LIN {X 0,Y 574.132,Z 514.669,A -85,B 0,C 180,E1 -2084.662,E2 -2084.662} C_VEL
LIN {X 0,Y 574.281,Z 500.292,A -85,B 0,C 180,E1 -2084.996,E2 -2084.996} C_VEL
LIN {X 0,Y 573.065,Z 493.165,A -85,B 0,C 180,E1 -2085.151,E2 -2085.151} C_VEL
LIN {X 0,Y 573.135,Z 485.279,A -85,B 0,C 180,E1 -2087.851,E2 -2087.851} C_VEL
LIN {X 0,Y 573.19,Z 477.793,A -85,B 0,C 180,E1 -2090.452,E2 -2090.452} C_VEL
LIN {X 0,Y 573.212,Z 470.196,A -85,B 0,C 180,E1 -2093.139,E2 -2093.139} C_VEL
LIN {X 0,Y 573.285,Z 462.82,A -85,B 0,C 180,E1 -2095.797,E2 -2095.797} C_VEL
LIN {X 0,Y 573.314,Z 455.113,A -85,B 0,C 180,E1 -2098.559,E2 -2098.559} C_VEL
LIN {X 0,Y 573.308,Z 448.157,A -85,B 0,C 180,E1 -2100.987,E2 -2100.987} C_VEL
LIN {X 0,Y 573.317,Z 439.853,A -85,B 0,C 180,E1 -2103.899,E2 -2103.899} C_VEL
LIN {X 0,Y 573.354,Z 431.271,A -85,B 0,C 180,E1 -2106.913,E2 -2106.913} C_VEL
LIN {X 0,Y 573.295,Z 427.699,A -85,B 0,C 180,E1 -2108.186,E2 -2108.186} C_VEL
LIN {X 0,Y 573.264,Z 427.702,A -85,B 0,C 180,E1 -2110.527,E2 -2110.527} C_VEL
LIN {X 0,Y 573.246,Z 427.701,A -85,B 0,C 180,E1 -2113.669,E2 -2113.669} C_VEL
LIN {X 0,Y 573.247,Z 427.703,A -85,B 0,C 180,E1 -2116.641,E2 -2116.641} C_VEL
LIN {X 0,Y 573.267,Z 427.705,A -85,B 0,C 180,E1 -2119.477,E2 -2119.477} C_VEL
LIN {X 0,Y 573.23,Z 427.703,A -85,B 0,C 180,E1 -2122.192,E2 -2122.192} C_VEL
LIN {X 0,Y 573.26,Z 427.706,A -85,B 0,C 180,E1 -2124.816,E2 -2124.816} C_VEL
LIN {X 0,Y 573.25,Z 427.701,A -85,B 0,C 180,E1 -2127.355,E2 -2127.355} C_VEL
LIN {X 0,Y 573.248,Z 427.705,A -85,B 0,C 180,E1 -2129.824,E2 -2129.824} C_VEL
LIN {X 0,Y 573.28,Z 427.697,A -85,B 0,C 180,E1 -2132.234,E2 -2132.234} C_VEL
LIN {X 0,Y 573.26,Z 427.706,A -85,B 0,C 180,E1 -2135.12,E2 -2135.12} C_VEL
LIN {X 0,Y 573.25,Z 427.699,A -85,B 0,C 180,E1 -2137.663,E2 -2137.663} C_VEL
LIN {X 0,Y 573.27,Z 427.701,A -85,B 0,C 180,E1 -2140.727,E2 -2140.727} C_VEL
LIN {X 0,Y 573.252,Z 427.704,A -85,B 0,C 180,E1 -2143.622,E2 -2143.622} C_VEL
LIN {X 0,Y 573.23,Z 427.703,A -85,B 0,C 180,E1 -2146.529,E2 -2146.529} C_VEL
LIN {X 0,Y 573.273,Z 427.7,A -85,B 0,C 180,E1 -2148.734,E2 -2148.734} C_VEL
LIN {X 0,Y 573.3,Z 427.693,A -85,B 0,C 180,E1 -2151.541,E2 -2151.541} C_VEL
LIN {X 0,Y 573.295,Z 427.7,A -85,B 0,C 180,E1 -2154.372,E2 -2154.372} C_VEL
LIN {X 0,Y 573.3,Z 427.698,A -85,B 0,C 180,E1 -2157.892,E2 -2157.892} C_VEL
LIN {X 0,Y 573.328,Z 427.692,A -85,B 0,C 180,E1 -2160.702,E2 -2160.702} C_VEL
LIN {X 0,Y 573.236,Z 427.699,A -85,B 0,C 180,E1 -2163.514,E2 -2163.514} C_VEL
LIN {X 0,Y 573.287,Z 427.695,A -85,B 0,C 180,E1 -2165.628,E2 -2165.628} C_VEL
LIN {X 0,Y 573.3,Z 427.696,A -85,B 0,C 180,E1 -2168.459,E2 -2168.459} C_VEL
LIN {X 0,Y 573.288,Z 427.696,A -85,B 0,C 180,E1 -2171.312,E2 -2171.312} C_VEL
LIN {X 0,Y 573.271,Z 427.698,A -85,B 0,C 180,E1 -2174.425,E2 -2174.425} C_VEL
LIN {X 0,Y 573.251,Z 427.7,A -85,B 0,C 180,E1 -2177.112,E2 -2177.112} C_VEL
LIN {X 0,Y 573.249,Z 427.705,A -85,B 0,C 180,E1 -2180.077,E2 -2180.077} C_VEL
LIN {X 0,Y 573.234,Z 427.705,A -85,B 0,C 180,E1 -2182.338,E2 -2182.338} C_VEL
LIN {X 0,Y 573.248,Z 427.708,A -85,B 0,C 180,E1 -2185.41,E2 -2185.41} C_VEL
LIN {X 0,Y 573.256,Z 427.699,A -85,B 0,C 180,E1 -2188.033,E2 -2188.033} C_VEL
LIN {X 0,Y 573.237,Z 427.706,A -85,B 0,C 180,E1 -2190.886,E2 -2190.886} C_VEL
LIN {X 0,Y 573.279,Z 427.698,A -85,B 0,C 180,E1 -2193.529,E2 -2193.529} C_VEL
LIN {X 0,Y 573.253,Z 427.704,A -85,B 0,C 180,E1 -2196.049,E2 -2196.049} C_VEL
LIN {X 0,Y 573.242,Z 427.702,A -85,B 0,C 180,E1 -2198.702,E2 -2198.702} C_VEL
LIN {X 0,Y 573.259,Z 427.7,A -85,B 0,C 180,E1 -2201.598,E2 -2201.598} C_VEL
LIN {X 0,Y 573.232,Z 427.708,A -85,B 0,C 180,E1 -2204.334,E2 -2204.334} C_VEL
LIN {X 0,Y 573.234,Z 427.703,A -85,B 0,C 180,E1 -2207.359,E2 -2207.359} C_VEL
LIN {X 0,Y 573.245,Z 427.702,A -85,B 0,C 180,E1 -2210.394,E2 -2210.394} C_VEL
LIN {X 0,Y 573.251,Z 427.707,A -85,B 0,C 180,E1 -2213.079,E2 -2213.079} C_VEL
LIN {X 0,Y 573.271,Z 427.701,A -85,B 0,C 180,E1 -2215.673,E2 -2215.673} C_VEL
LIN {X 0,Y 573.301,Z 427.855,A -85,B 0,C 180,E1 -2216.679,E2 -2216.679} C_VEL
LIN {X 0,Y 573.955,Z 432.32,A -85,B 0,C 180,E1 -2217.952,E2 -2217.952} C_VEL
LIN {X 0,Y 573.773,Z 442.67,A -85,B 0,C 180,E1 -2220.664,E2 -2220.664} C_VEL
LIN {X 0,Y 573.669,Z 453.5,A -85,B 0,C 180,E1 -2223.421,E2 -2223.421} C_VEL
LIN {X 0,Y 573.507,Z 464.501,A -85,B 0,C 180,E1 -2226.148,E2 -2226.148} C_VEL
LIN {X 0,Y 573.373,Z 476.989,A -85,B 0,C 180,E1 -2229.179,E2 -2229.179} C_VEL
LIN {X 0,Y 573.305,Z 489.478,A -85,B 0,C 180,E1 -2232.155,E2 -2232.155} C_VEL
LIN {X 0,Y 573.22,Z 501.089,A -85,B 0,C 180,E1 -2234.876,E2 -2234.876} C_VEL
LIN {X 0,Y 574.273,Z 507.817,A -85,B 0,C 180,E1 -2235.005,E2 -2235.005} C_VEL
LIN {X 0,Y 574.185,Z 522.276,A -85,B 0,C 180,E1 -2235.316,E2 -2235.316} C_VEL
LIN {X 0,Y 574.055,Z 536.338,A -85,B 0,C 180,E1 -2235.772,E2 -2235.772} C_VEL
LIN {X 0,Y 573.93,Z 549.901,A -85,B 0,C 180,E1 -2236.367,E2 -2236.367} C_VEL
LIN {X 0,Y 573.716,Z 562.7,A -85,B 0,C 180,E1 -2237.083,E2 -2237.083} C_VEL
LIN {X 0,Y 573.571,Z 575.491,A -85,B 0,C 180,E1 -2237.978,E2 -2237.978} C_VEL
LIN {X 0,Y 573.448,Z 586.864,A -85,B 0,C 180,E1 -2238.956,E2 -2238.956} C_VEL
LIN {X 0,Y 573.268,Z 596.342,A -85,B 0,C 180,E1 -2239.94,E2 -2239.94} C_VEL
LIN {X 0,Y 573.19,Z 604.92,A -85,B 0,C 180,E1 -2241.007,E2 -2241.007} C_VEL
LIN {X 0,Y 573.111,Z 613.121,A -85,B 0,C 180,E1 -2242.249,E2 -2242.249} C_VEL
LIN {X 0,Y 573.035,Z 619.452,A -85,B 0,C 180,E1 -2243.427,E2 -2243.427} C_VEL
LIN {X 0,Y 573.001,Z 624.965,A -85,B 0,C 180,E1 -2244.723,E2 -2244.723} C_VEL
LIN {X 0,Y 573.028,Z 628.445,A -85,B 0,C 180,E1 -2245.781,E2 -2245.781} C_VEL
LIN {X 0,Y 572.956,Z 631.833,A -85,B 0,C 180,E1 -2247.189,E2 -2247.189} C_VEL
LIN {X 0,Y 572.941,Z 633.833,A -85,B 0,C 180,E1 -2248.595,E2 -2248.595} C_VEL
LIN {X 0,Y 572.937,Z 634.5,A -85,B 0,C 180,E1 -2250.001,E2 -2250.001} C_VEL
LIN {X 0,Y 572.941,Z 633.832,A -85,B 0,C 180,E1 -2251.407,E2 -2251.407} C_VEL
LIN {X 0,Y 572.956,Z 631.831,A -85,B 0,C 180,E1 -2252.813,E2 -2252.813} C_VEL
LIN {X 0,Y 573.028,Z 628.441,A -85,B 0,C 180,E1 -2254.221,E2 -2254.221} C_VEL
LIN {X 0,Y 573.055,Z 623.564,A -85,B 0,C 180,E1 -2255.631,E2 -2255.631} C_VEL
LIN {X 0,Y 573.059,Z 618.849,A -85,B 0,C 180,E1 -2256.693,E2 -2256.693} C_VEL
LIN {X 0,Y 573.126,Z 612.032,A -85,B 0,C 180,E1 -2257.93,E2 -2257.93} C_VEL
LIN {X 0,Y 573.226,Z 603.553,A -85,B 0,C 180,E1 -2259.172,E2 -2259.172} C_VEL
LIN {X 0,Y 573.305,Z 594.7,A -85,B 0,C 180,E1 -2260.24,E2 -2260.24} C_VEL
LIN {X 0,Y 573.464,Z 583.983,A -85,B 0,C 180,E1 -2261.309,E2 -2261.309} C_VEL
LIN {X 0,Y 573.622,Z 573.133,A -85,B 0,C 180,E1 -2262.202,E2 -2262.202} C_VEL
LIN {X 0,Y 573.736,Z 561.247,A -85,B 0,C 180,E1 -2263.009,E2 -2263.009} C_VEL
LIN {X 0,Y 573.95,Z 548.078,A -85,B 0,C 180,E1 -2263.725,E2 -2263.725} C_VEL
LIN {X 0,Y 574.08,Z 534.798,A -85,B 0,C 180,E1 -2264.285,E2 -2264.285} C_VEL
LIN {X 0,Y 574.206,Z 520.732,A -85,B 0,C 180,E1 -2264.722,E2 -2264.722} C_VEL
LIN {X 0,Y 574.197,Z 506.39,A -85,B 0,C 180,E1 -2265.019,E2 -2265.019} C_VEL
LIN {X 0,Y 573.209,Z 501.081,A -85,B 0,C 180,E1 -2265.126,E2 -2265.126} C_VEL
LIN {X 0,Y 573.307,Z 489.47,A -85,B 0,C 180,E1 -2267.847,E2 -2267.847} C_VEL
LIN {X 0,Y 573.373,Z 476.982,A -85,B 0,C 180,E1 -2270.822,E2 -2270.822} C_VEL
LIN {X 0,Y 573.516,Z 465.991,A -85,B 0,C 180,E1 -2273.486,E2 -2273.486} C_VEL
LIN {X 0,Y 573.613,Z 455.126,A -85,B 0,C 180,E1 -2276.173,E2 -2276.173} C_VEL
LIN {X 0,Y 573.767,Z 445.866,A -85,B 0,C 180,E1 -2278.536,E2 -2278.536} C_VEL
LIN {X 0,Y 573.946,Z 436.55,A -85,B 0,C 180,E1 -2281.001,E2 -2281.001} C_VEL
LIN {X 0,Y 574.002,Z 431.778,A -85,B 0,C 180,E1 -2282.347,E2 -2282.347} C_VEL
LIN {X 0,Y 573.275,Z 427.703,A -85,B 0,C 180,E1 -2283.693,E2 -2283.693} C_VEL
LIN {X 0,Y 573.244,Z 427.708,A -85,B 0,C 180,E1 -2286.05,E2 -2286.05} C_VEL
LIN {X 0,Y 573.253,Z 427.705,A -85,B 0,C 180,E1 -2288.701,E2 -2288.701} C_VEL
LIN {X 0,Y 573.233,Z 427.707,A -85,B 0,C 180,E1 -2291.458,E2 -2291.458} C_VEL
LIN {X 0,Y 573.229,Z 427.707,A -85,B 0,C 180,E1 -2294.335,E2 -2294.335} C_VEL
LIN {X 0,Y 573.252,Z 427.705,A -85,B 0,C 180,E1 -2296.642,E2 -2296.642} C_VEL
LIN {X 0,Y 573.249,Z 427.707,A -85,B 0,C 180,E1 -2299.475,E2 -2299.475} C_VEL
LIN {X 0,Y 573.239,Z 427.71,A -85,B 0,C 180,E1 -2302.193,E2 -2302.193} C_VEL
LIN {X 0,Y 573.313,Z 427.8,A -85,B 0,C 180,E1 -2304.551,E2 -2304.551} C_VEL
LIN {X 0,Y 573.264,Z 433.787,A -85,B 0,C 180,E1 -2307.356,E2 -2307.356} C_VEL
LIN {X 0,Y 573.239,Z 440.605,A -85,B 0,C 180,E1 -2310.514,E2 -2310.514} C_VEL
LIN {X 0,Y 573.167,Z 446.058,A -85,B 0,C 180,E1 -2313.02,E2 -2313.02} C_VEL
LIN {X 0,Y 573.161,Z 451.002,A -85,B 0,C 180,E1 -2315.361,E2 -2315.361} C_VEL
LIN {X 0,Y 573.094,Z 457.867,A -85,B 0,C 180,E1 -2318.414,E2 -2318.414} C_VEL
LIN {X 0,Y 573.064,Z 464.731,A -85,B 0,C 180,E1 -2321.406,E2 -2321.406} C_VEL
LIN {X 0,Y 573.047,Z 469.879,A -85,B 0,C 180,E1 -2323.616,E2 -2323.616} C_VEL
LIN {X 0,Y 573.049,Z 475.028,A -85,B 0,C 180,E1 -2325.801,E2 -2325.801} C_VEL
LIN {X 0,Y 573.015,Z 479.212,A -85,B 0,C 180,E1 -2327.561,E2 -2327.561} C_VEL
LIN {X 0,Y 573.855,Z 486.016,A -85,B 0,C 180,E1 -2327.714,E2 -2327.714} C_VEL
LIN {X 0,Y 573.738,Z 498.671,A -85,B 0,C 180,E1 -2328.071,E2 -2328.071} C_VEL
LIN {X 0,Y 573.604,Z 511.366,A -85,B 0,C 180,E1 -2328.578,E2 -2328.578} C_VEL
LIN {X 0,Y 573.544,Z 522.177,A -85,B 0,C 180,E1 -2329.147,E2 -2329.147} C_VEL
LIN {X 0,Y 573.441,Z 532.835,A -85,B 0,C 180,E1 -2329.853,E2 -2329.853} C_VEL
LIN {X 0,Y 573.321,Z 542.609,A -85,B 0,C 180,E1 -2330.652,E2 -2330.652} C_VEL
LIN {X 0,Y 573.235,Z 551.501,A -85,B 0,C 180,E1 -2331.54,E2 -2331.54} C_VEL
LIN {X 0,Y 573.126,Z 560.184,A -85,B 0,C 180,E1 -2332.602,E2 -2332.602} C_VEL
LIN {X 0,Y 573.049,Z 567.111,A -85,B 0,C 180,E1 -2333.663,E2 -2333.663} C_VEL
LIN {X 0,Y 573.009,Z 572.659,A -85,B 0,C 180,E1 -2334.722,E2 -2334.722} C_VEL
LIN {X 0,Y 573.031,Z 577.019,A -85,B 0,C 180,E1 -2335.78,E2 -2335.78} C_VEL
LIN {X 0,Y 573.023,Z 579.323,A -85,B 0,C 180,E1 -2336.484,E2 -2336.484} C_VEL
LIN {X 0,Y 572.959,Z 581.2,A -85,B 0,C 180,E1 -2337.188,E2 -2337.188} C_VEL
LIN {X 0,Y 572.938,Z 582.628,A -85,B 0,C 180,E1 -2337.891,E2 -2337.891} C_VEL
LIN {X 0,Y 572.941,Z 584.255,A -85,B 0,C 180,E1 -2339.297,E2 -2339.297} C_VEL
LIN {X 0,Y 572.938,Z 584.496,A -85,B 0,C 180,E1 -2340,E2 -2340} C_VEL
LIN {X 0,Y 572.941,Z 584.314,A -85,B 0,C 180,E1 -2340.703,E2 -2340.703} C_VEL
LIN {X 0,Y 572.937,Z 582.771,A -85,B 0,C 180,E1 -2342.109,E2 -2342.109} C_VEL
LIN {X 0,Y 572.96,Z 581.409,A -85,B 0,C 180,E1 -2342.812,E2 -2342.812} C_VEL
LIN {X 0,Y 573.015,Z 578.532,A -85,B 0,C 180,E1 -2343.868,E2 -2343.868} C_VEL
LIN {X 0,Y 572.963,Z 574.631,A -85,B 0,C 180,E1 -2344.926,E2 -2344.926} C_VEL
LIN {X 0,Y 573.073,Z 569.599,A -85,B 0,C 180,E1 -2345.984,E2 -2345.984} C_VEL
LIN {X 0,Y 573.084,Z 563.275,A -85,B 0,C 180,E1 -2347.044,E2 -2347.044} C_VEL
LIN {X 0,Y 573.175,Z 555.354,A -85,B 0,C 180,E1 -2348.106,E2 -2348.106} C_VEL
LIN {X 0,Y 573.287,Z 545.505,A -85,B 0,C 180,E1 -2349.17,E2 -2349.17} C_VEL
LIN {X 0,Y 573.412,Z 535.182,A -85,B 0,C 180,E1 -2350.059,E2 -2350.059} C_VEL
LIN {X 0,Y 573.509,Z 523.592,A -85,B 0,C 180,E1 -2350.857,E2 -2350.857} C_VEL
LIN {X 0,Y 573.642,Z 512.017,A -85,B 0,C 180,E1 -2351.482,E2 -2351.482} C_VEL
LIN {X 0,Y 573.729,Z 500.106,A -85,B 0,C 180,E1 -2351.97,E2 -2351.97} C_VEL
LIN {X 0,Y 573.859,Z 486.938,A -85,B 0,C 180,E1 -2352.353,E2 -2352.353} C_VEL
LIN {X 0,Y 573.47,Z 482.233,A -85,B 0,C 180,E1 -2352.461,E2 -2352.461} C_VEL
LIN {X 0,Y 573.01,Z 479.211,A -85,B 0,C 180,E1 -2352.529,E2 -2352.529} C_VEL
LIN {X 0,Y 573.05,Z 473.524,A -85,B 0,C 180,E1 -2354.925,E2 -2354.925} C_VEL
LIN {X 0,Y 573.062,Z 466.656,A -85,B 0,C 180,E1 -2357.854,E2 -2357.854} C_VEL
LIN {X 0,Y 573.069,Z 463.772,A -85,B 0,C 180,E1 -2359.099,E2 -2359.099} C_VEL
LIN {X 0,Y 572.427,Z 462.503,A -85,B 0,C 180,E1 -2359.672,E2 -2359.672} C_VEL
LIN {X 0,Y 569.575,Z 460.607,A -85,B 0,C 180,E1 -2360.606,E2 -2360.606} C_VEL
LIN {X 0,Y 567.148,Z 459.117,A -85,B 0,C 180,E1 -2361.358,E2 -2361.358} C_VEL
LIN {X 0,Y 566.103,Z 457.91,A -85,B 0,C 180,E1 -2361.938,E2 -2361.938} C_VEL
LIN {X 0,Y 566.017,Z 457.48,A -85,B 0,C 180,E1 -2362.133,E2 -2362.133} C_VEL
LIN {X 0,Y 566.079,Z 451.198,A -85,B 0,C 180,E1 -2364.999,E2 -2364.999} C_VEL
LIN {X 0,Y 566.104,Z 446.133,A -85,B 0,C 180,E1 -2367.345,E2 -2367.345} C_VEL
LIN {X 0,Y 566.17,Z 440.975,A -85,B 0,C 180,E1 -2369.771,E2 -2369.771} C_VEL
LIN {X 0,Y 566.218,Z 435.4,A -85,B 0,C 180,E1 -2372.431,E2 -2372.431} C_VEL
LIN {X 0,Y 566.268,Z 430.126,A -85,B 0,C 180,E1 -2375.001,E2 -2375.001} C_VEL
LIN {X 0,Y 566.25,Z 428.579,A -85,B 0,C 180,E1 -2375.875,E2 -2375.875} C_VEL
LIN {X 0,Y 566.213,Z 428.584,A -85,B 0,C 180,E1 -2378.558,E2 -2378.558} C_VEL
LIN {X 0,Y 566.188,Z 428.585,A -85,B 0,C 180,E1 -2381.139,E2 -2381.139} C_VEL
LIN {X 0,Y 566.207,Z 428.584,A -85,B 0,C 180,E1 -2384.035,E2 -2384.035} C_VEL
LIN {X 0,Y 566.206,Z 428.586,A -85,B 0,C 180,E1 -2387.083,E2 -2387.083} C_VEL
LIN {X 0,Y 566.226,Z 428.582,A -85,B 0,C 180,E1 -2390.313,E2 -2390.313} C_VEL
LIN {X 0,Y 566.269,Z 428.677,A -85,B 0,C 180,E1 -2391.926,E2 -2391.926} C_VEL
LIN {X 0,Y 566.32,Z 435.595,A -85,B 0,C 180,E1 -2394.319,E2 -2394.319} C_VEL
LIN {X 0,Y 566.316,Z 442.828,A -85,B 0,C 180,E1 -2396.903,E2 -2396.903} C_VEL
LIN {X 0,Y 566.298,Z 451.061,A -85,B 0,C 180,E1 -2399.826,E2 -2399.826} C_VEL
LIN {X 0,Y 566.263,Z 459.132,A -85,B 0,C 180,E1 -2402.663,E2 -2402.663} C_VEL
LIN {X 0,Y 566.246,Z 466.845,A -85,B 0,C 180,E1 -2405.43,E2 -2405.43} C_VEL
LIN {X 0,Y 566.183,Z 475.585,A -85,B 0,C 180,E1 -2408.587,E2 -2408.587} C_VEL
LIN {X 0,Y 566.086,Z 483.945,A -85,B 0,C 180,E1 -2411.543,E2 -2411.543} C_VEL
LIN {X 0,Y 566.017,Z 492.496,A -85,B 0,C 180,E1 -2414.516,E2 -2414.516} C_VEL
LIN {X 0,Y 566.013,Z 493.383,A -85,B 0,C 180,E1 -2414.758,E2 -2414.758} C_VEL
LIN {X 0,Y 567.439,Z 501.104,A -85,B 0,C 180,E1 -2414.924,E2 -2414.924} C_VEL
LIN {X 0,Y 567.276,Z 516.71,A -85,B 0,C 180,E1 -2415.31,E2 -2415.31} C_VEL
LIN {X 0,Y 567.102,Z 529.875,A -85,B 0,C 180,E1 -2415.786,E2 -2415.786} C_VEL
LIN {X 0,Y 566.961,Z 542.498,A -85,B 0,C 180,E1 -2416.377,E2 -2416.377} C_VEL
LIN {X 0,Y 566.741,Z 554.822,A -85,B 0,C 180,E1 -2417.101,E2 -2417.101} C_VEL
LIN {X 0,Y 566.578,Z 566.047,A -85,B 0,C 180,E1 -2417.917,E2 -2417.917} C_VEL
LIN {X 0,Y 566.434,Z 576.759,A -85,B 0,C 180,E1 -2418.858,E2 -2418.858} C_VEL
LIN {X 0,Y 566.266,Z 585.882,A -85,B 0,C 180,E1 -2419.812,E2 -2419.812} C_VEL
LIN {X 0,Y 566.152,Z 594.566,A -85,B 0,C 180,E1 -2420.892,E2 -2420.892} C_VEL
LIN {X 0,Y 566.061,Z 602.827,A -85,B 0,C 180,E1 -2422.15,E2 -2422.15} C_VEL
LIN {X 0,Y 565.968,Z 609.557,A -85,B 0,C 180,E1 -2423.421,E2 -2423.421} C_VEL
LIN {X 0,Y 565.928,Z 614.762,A -85,B 0,C 180,E1 -2424.655,E2 -2424.655} C_VEL
LIN {X 0,Y 565.957,Z 618.292,A -85,B 0,C 180,E1 -2425.726,E2 -2425.726} C_VEL
LIN {X 0,Y 565.875,Z 621.747,A -85,B 0,C 180,E1 -2427.152,E2 -2427.152} C_VEL
LIN {X 0,Y 565.844,Z 623.787,A -85,B 0,C 180,E1 -2428.576,E2 -2428.576} C_VEL
LIN {X 0,Y 565.838,Z 624.461,A -85,B 0,C 180,E1 -2429.999,E2 -2429.999} C_VEL
LIN {X 0,Y 565.841,Z 623.857,A -85,B 0,C 180,E1 -2431.423,E2 -2431.423} C_VEL
LIN {X 0,Y 565.873,Z 621.932,A -85,B 0,C 180,E1 -2432.847,E2 -2432.847} C_VEL
LIN {X 0,Y 565.958,Z 618.564,A -85,B 0,C 180,E1 -2434.272,E2 -2434.272} C_VEL
LIN {X 0,Y 565.929,Z 615.115,A -85,B 0,C 180,E1 -2435.343,E2 -2435.343} C_VEL
LIN {X 0,Y 565.966,Z 609.99,A -85,B 0,C 180,E1 -2436.577,E2 -2436.577} C_VEL
LIN {X 0,Y 566.059,Z 603.344,A -85,B 0,C 180,E1 -2437.849,E2 -2437.849} C_VEL
LIN {X 0,Y 566.145,Z 595.247,A -85,B 0,C 180,E1 -2439.106,E2 -2439.106} C_VEL
LIN {X 0,Y 566.246,Z 586.707,A -85,B 0,C 180,E1 -2440.186,E2 -2440.186} C_VEL
LIN {X 0,Y 566.407,Z 577.698,A -85,B 0,C 180,E1 -2441.142,E2 -2441.142} C_VEL
LIN {X 0,Y 566.516,Z 568.249,A -85,B 0,C 180,E1 -2441.992,E2 -2441.992} C_VEL
LIN {X 0,Y 566.712,Z 557.462,A -85,B 0,C 180,E1 -2442.806,E2 -2442.806} C_VEL
LIN {X 0,Y 566.881,Z 545.87,A -85,B 0,C 180,E1 -2443.532,E2 -2443.532} C_VEL
LIN {X 0,Y 567.076,Z 532.095,A -85,B 0,C 180,E1 -2444.213,E2 -2444.213} C_VEL
LIN {X 0,Y 567.228,Z 518.993,A -85,B 0,C 180,E1 -2444.706,E2 -2444.706} C_VEL
LIN {X 0,Y 567.378,Z 506.474,A -85,B 0,C 180,E1 -2445.052,E2 -2445.052} C_VEL
LIN {X 0,Y 567.2,Z 499.242,A -85,B 0,C 180,E1 -2445.204,E2 -2445.204} C_VEL
LIN {X 0,Y 566.006,Z 493.163,A -85,B 0,C 180,E1 -2445.344,E2 -2445.344} C_VEL
LIN {X 0,Y 566.063,Z 485.277,A -85,B 0,C 180,E1 -2448.082,E2 -2448.082} C_VEL
LIN {X 0,Y 566.132,Z 477.791,A -85,B 0,C 180,E1 -2450.719,E2 -2450.719} C_VEL
LIN {X 0,Y 566.214,Z 469.235,A -85,B 0,C 180,E1 -2453.79,E2 -2453.79} C_VEL
LIN {X 0,Y 566.278,Z 461.252,A -85,B 0,C 180,E1 -2456.673,E2 -2456.673} C_VEL
LIN {X 0,Y 566.316,Z 452.498,A -85,B 0,C 180,E1 -2459.761,E2 -2459.761} C_VEL
LIN {X 0,Y 566.268,Z 444.946,A -85,B 0,C 180,E1 -2462.44,E2 -2462.44} C_VEL
LIN {X 0,Y 566.307,Z 437.755,A -85,B 0,C 180,E1 -2465.007,E2 -2465.007} C_VEL
LIN {X 0,Y 566.374,Z 430.788,A -85,B 0,C 180,E1 -2467.446,E2 -2467.446} C_VEL
LIN {X 0,Y 566.24,Z 428.578,A -85,B 0,C 180,E1 -2468.244,E2 -2468.244} C_VEL
LIN {X 0,Y 566.207,Z 428.583,A -85,B 0,C 180,E1 -2471.135,E2 -2471.135} C_VEL
LIN {X 0,Y 566.194,Z 428.583,A -85,B 0,C 180,E1 -2474.034,E2 -2474.034} C_VEL
LIN {X 0,Y 566.208,Z 428.578,A -85,B 0,C 180,E1 -2477.08,E2 -2477.08} C_VEL
LIN {X 0,Y 566.22,Z 428.58,A -85,B 0,C 180,E1 -2479.802,E2 -2479.802} C_VEL
LIN {X 0,Y 566.192,Z 428.581,A -85,B 0,C 180,E1 -2482.598,E2 -2482.598} C_VEL
LIN {X 0,Y 566.213,Z 428.578,A -85,B 0,C 180,E1 -2485.182,E2 -2485.182} C_VEL
LIN {X 0,Y 566.229,Z 428.577,A -85,B 0,C 180,E1 -2487.743,E2 -2487.743} C_VEL
LIN {X 0,Y 566.22,Z 428.579,A -85,B 0,C 180,E1 -2490.323,E2 -2490.323} C_VEL
LIN {X 0,Y 566.226,Z 428.581,A -85,B 0,C 180,E1 -2493.334,E2 -2493.334} C_VEL
LIN {X 0,Y 566.196,Z 428.579,A -85,B 0,C 180,E1 -2495.819,E2 -2495.819} C_VEL
LIN {X 0,Y 566.208,Z 428.581,A -85,B 0,C 180,E1 -2498.902,E2 -2498.902} C_VEL
LIN {X 0,Y 566.206,Z 428.578,A -85,B 0,C 180,E1 -2501.172,E2 -2501.172} C_VEL
LIN {X 0,Y 566.214,Z 428.579,A -85,B 0,C 180,E1 -2503.412,E2 -2503.412} C_VEL
LIN {X 0,Y 566.192,Z 428.58,A -85,B 0,C 180,E1 -2506.359,E2 -2506.359} C_VEL
LIN {X 0,Y 566.265,Z 428.572,A -85,B 0,C 180,E1 -2508.654,E2 -2508.654} C_VEL
LIN {X 0,Y 566.241,Z 428.573,A -85,B 0,C 180,E1 -2511.434,E2 -2511.434} C_VEL
LIN {X 0,Y 566.263,Z 428.577,A -85,B 0,C 180,E1 -2514.302,E2 -2514.302} C_VEL
LIN {X 0,Y 566.271,Z 428.574,A -85,B 0,C 180,E1 -2517.866,E2 -2517.866} C_VEL
LIN {X 0,Y 566.298,Z 428.568,A -85,B 0,C 180,E1 -2520.711,E2 -2520.711} C_VEL
LIN {X 0,Y 566.272,Z 428.574,A -85,B 0,C 180,E1 -2522.846,E2 -2522.846} C_VEL
LIN {X 0,Y 566.254,Z 428.571,A -85,B 0,C 180,E1 -2525.698,E2 -2525.698} C_VEL
LIN {X 0,Y 566.241,Z 428.574,A -85,B 0,C 180,E1 -2528.565,E2 -2528.565} C_VEL
LIN {X 0,Y 566.24,Z 428.576,A -85,B 0,C 180,E1 -2531.454,E2 -2531.454} C_VEL
LIN {X 0,Y 566.223,Z 428.577,A -85,B 0,C 180,E1 -2534.507,E2 -2534.507} C_VEL
LIN {X 0,Y 566.196,Z 428.577,A -85,B 0,C 180,E1 -2537.332,E2 -2537.332} C_VEL
LIN {X 0,Y 566.211,Z 428.583,A -85,B 0,C 180,E1 -2540.337,E2 -2540.337} C_VEL
LIN {X 0,Y 566.181,Z 428.584,A -85,B 0,C 180,E1 -2543.404,E2 -2543.404} C_VEL
LIN {X 0,Y 566.217,Z 428.58,A -85,B 0,C 180,E1 -2545.749,E2 -2545.749} C_VEL
LIN {X 0,Y 566.199,Z 428.579,A -85,B 0,C 180,E1 -2548.204,E2 -2548.204} C_VEL
LIN {X 0,Y 566.187,Z 428.588,A -85,B 0,C 180,E1 -2550.592,E2 -2550.592} C_VEL
LIN {X 0,Y 566.221,Z 428.576,A -85,B 0,C 180,E1 -2553.102,E2 -2553.102} C_VEL
LIN {X 0,Y 566.204,Z 428.584,A -85,B 0,C 180,E1 -2555.689,E2 -2555.689} C_VEL
LIN {X 0,Y 566.208,Z 428.578,A -85,B 0,C 180,E1 -2558.56,E2 -2558.56} C_VEL
LIN {X 0,Y 566.214,Z 428.583,A -85,B 0,C 180,E1 -2561.136,E2 -2561.136} C_VEL
LIN {X 0,Y 566.194,Z 428.581,A -85,B 0,C 180,E1 -2564.036,E2 -2564.036} C_VEL
LIN {X 0,Y 566.195,Z 428.58,A -85,B 0,C 180,E1 -2567.084,E2 -2567.084} C_VEL
LIN {X 0,Y 566.222,Z 428.582,A -85,B 0,C 180,E1 -2569.804,E2 -2569.804} C_VEL
LIN {X 0,Y 566.194,Z 428.581,A -85,B 0,C 180,E1 -2572.6,E2 -2572.6} C_VEL
LIN {X 0,Y 566.219,Z 428.583,A -85,B 0,C 180,E1 -2575.184,E2 -2575.184} C_VEL
LIN {X 0,Y 566.251,Z 428.637,A -85,B 0,C 180,E1 -2576.406,E2 -2576.406} C_VEL
LIN {X 0,Y 567.021,Z 433.425,A -85,B 0,C 180,E1 -2577.795,E2 -2577.795} C_VEL
LIN {X 0,Y 566.875,Z 442.691,A -85,B 0,C 180,E1 -2580.271,E2 -2580.271} C_VEL
LIN {X 0,Y 566.681,Z 454.21,A -85,B 0,C 180,E1 -2583.246,E2 -2583.246} C_VEL
LIN {X 0,Y 566.532,Z 464.501,A -85,B 0,C 180,E1 -2585.836,E2 -2585.836} C_VEL
LIN {X 0,Y 566.4,Z 475.435,A -85,B 0,C 180,E1 -2588.531,E2 -2588.531} C_VEL
LIN {X 0,Y 566.288,Z 487.917,A -85,B 0,C 180,E1 -2591.551,E2 -2591.551} C_VEL
LIN {X 0,Y 566.161,Z 500.796,A -85,B 0,C 180,E1 -2594.614,E2 -2594.614} C_VEL
LIN {X 0,Y 566.175,Z 501.089,A -85,B 0,C 180,E1 -2594.684,E2 -2594.684} C_VEL
LIN {X 0,Y 567.42,Z 508.702,A -85,B 0,C 180,E1 -2594.833,E2 -2594.833} C_VEL
LIN {X 0,Y 567.316,Z 522.984,A -85,B 0,C 180,E1 -2595.154,E2 -2595.154} C_VEL
LIN {X 0,Y 567.168,Z 536.43,A -85,B 0,C 180,E1 -2595.599,E2 -2595.599} C_VEL
LIN {X 0,Y 567.015,Z 549.9,A -85,B 0,C 180,E1 -2596.197,E2 -2596.197} C_VEL
LIN {X 0,Y 566.766,Z 562.698,A -85,B 0,C 180,E1 -2596.922,E2 -2596.922} C_VEL
LIN {X 0,Y 566.612,Z 574.329,A -85,B 0,C 180,E1 -2597.737,E2 -2597.737} C_VEL
LIN {X 0,Y 566.39,Z 584.525,A -85,B 0,C 180,E1 -2598.598,E2 -2598.598} C_VEL
LIN {X 0,Y 566.294,Z 594.716,A -85,B 0,C 180,E1 -2599.634,E2 -2599.634} C_VEL
LIN {X 0,Y 566.18,Z 603.566,A -85,B 0,C 180,E1 -2600.715,E2 -2600.715} C_VEL
LIN {X 0,Y 566.046,Z 612.043,A -85,B 0,C 180,E1 -2601.972,E2 -2601.972} C_VEL
LIN {X 0,Y 565.965,Z 619.806,A -85,B 0,C 180,E1 -2603.423,E2 -2603.423} C_VEL
LIN {X 0,Y 565.928,Z 624.965,A -85,B 0,C 180,E1 -2604.657,E2 -2604.657} C_VEL
LIN {X 0,Y 565.956,Z 628.445,A -85,B 0,C 180,E1 -2605.728,E2 -2605.728} C_VEL
LIN {X 0,Y 565.874,Z 631.833,A -85,B 0,C 180,E1 -2607.153,E2 -2607.153} C_VEL
LIN {X 0,Y 565.84,Z 633.833,A -85,B 0,C 180,E1 -2608.577,E2 -2608.577} C_VEL
LIN {X 0,Y 565.837,Z 634.5,A -85,B 0,C 180,E1 -2610.001,E2 -2610.001} C_VEL
LIN {X 0,Y 565.84,Z 633.832,A -85,B 0,C 180,E1 -2611.424,E2 -2611.424} C_VEL
LIN {X 0,Y 565.875,Z 631.832,A -85,B 0,C 180,E1 -2612.848,E2 -2612.848} C_VEL
LIN {X 0,Y 565.956,Z 628.442,A -85,B 0,C 180,E1 -2614.274,E2 -2614.274} C_VEL
LIN {X 0,Y 565.982,Z 623.565,A -85,B 0,C 180,E1 -2615.702,E2 -2615.702} C_VEL
LIN {X 0,Y 565.993,Z 619.04,A -85,B 0,C 180,E1 -2616.74,E2 -2616.74} C_VEL
LIN {X 0,Y 566.048,Z 612.032,A -85,B 0,C 180,E1 -2618.03,E2 -2618.03} C_VEL
LIN {X 0,Y 566.177,Z 603.552,A -85,B 0,C 180,E1 -2619.287,E2 -2619.287} C_VEL
LIN {X 0,Y 566.295,Z 594.7,A -85,B 0,C 180,E1 -2620.368,E2 -2620.368} C_VEL
LIN {X 0,Y 566.487,Z 583.982,A -85,B 0,C 180,E1 -2621.45,E2 -2621.45} C_VEL
LIN {X 0,Y 566.64,Z 573.132,A -85,B 0,C 180,E1 -2622.355,E2 -2622.355} C_VEL
LIN {X 0,Y 566.776,Z 561.246,A -85,B 0,C 180,E1 -2623.171,E2 -2623.171} C_VEL
LIN {X 0,Y 567.048,Z 548.079,A -85,B 0,C 180,E1 -2623.895,E2 -2623.895} C_VEL
LIN {X 0,Y 567.199,Z 535.028,A -85,B 0,C 180,E1 -2624.454,E2 -2624.454} C_VEL
LIN {X 0,Y 567.352,Z 521.169,A -85,B 0,C 180,E1 -2624.893,E2 -2624.893} C_VEL
LIN {X 0,Y 567.334,Z 507.288,A -85,B 0,C 180,E1 -2625.191,E2 -2625.191} C_VEL
LIN {X 0,Y 566.165,Z 501.081,A -85,B 0,C 180,E1 -2625.318,E2 -2625.318} C_VEL
LIN {X 0,Y 566.276,Z 489.47,A -85,B 0,C 180,E1 -2628.076,E2 -2628.076} C_VEL
LIN {X 0,Y 566.39,Z 476.982,A -85,B 0,C 180,E1 -2631.091,E2 -2631.091} C_VEL
LIN {X 0,Y 566.528,Z 466.054,A -85,B 0,C 180,E1 -2633.778,E2 -2633.778} C_VEL
LIN {X 0,Y 566.663,Z 455.064,A -85,B 0,C 180,E1 -2636.519,E2 -2636.519} C_VEL
LIN {X 0,Y 566.881,Z 444.352,A -85,B 0,C 180,E1 -2639.322,E2 -2639.322} C_VEL
LIN {X 0,Y 567.146,Z 433.994,A -85,B 0,C 180,E1 -2642.199,E2 -2642.199} C_VEL
LIN {X 0,Y 566.223,Z 428.583,A -85,B 0,C 180,E1 -2644.009,E2 -2644.009} C_VEL
LIN {X 0,Y 566.213,Z 428.581,A -85,B 0,C 180,E1 -2646.57,E2 -2646.57} C_VEL
LIN {X 0,Y 566.217,Z 428.58,A -85,B 0,C 180,E1 -2649.686,E2 -2649.686} C_VEL
LIN {X 0,Y 566.193,Z 428.586,A -85,B 0,C 180,E1 -2652.09,E2 -2652.09} C_VEL
LIN {X 0,Y 566.174,Z 428.588,A -85,B 0,C 180,E1 -2655.037,E2 -2655.037} C_VEL
LIN {X 0,Y 566.216,Z 428.584,A -85,B 0,C 180,E1 -2657.913,E2 -2657.913} C_VEL
LIN {X 0,Y 566.216,Z 428.584,A -85,B 0,C 180,E1 -2660.726,E2 -2660.726} C_VEL
LIN {X 0,Y 566.209,Z 428.585,A -85,B 0,C 180,E1 -2663.786,E2 -2663.786} C_VEL
LIN {X 0,Y 566.231,Z 428.663,A -85,B 0,C 180,E1 -2664.405,E2 -2664.405} C_VEL
LIN {X 0,Y 566.281,Z 432.504,A -85,B 0,C 180,E1 -2666.256,E2 -2666.256} C_VEL
LIN {X 0,Y 566.193,Z 438.122,A -85,B 0,C 180,E1 -2668.924,E2 -2668.924} C_VEL
LIN {X 0,Y 566.191,Z 444.411,A -85,B 0,C 180,E1 -2671.856,E2 -2671.856} C_VEL
LIN {X 0,Y 566.114,Z 449.512,A -85,B 0,C 180,E1 -2674.246,E2 -2674.246} C_VEL
LIN {X 0,Y 566.054,Z 454.784,A -85,B 0,C 180,E1 -2676.747,E2 -2676.747} C_VEL
LIN {X 0,Y 566.004,Z 461.3,A -85,B 0,C 180,E1 -2679.655,E2 -2679.655} C_VEL
LIN {X 0,Y 565.989,Z 466.449,A -85,B 0,C 180,E1 -2681.915,E2 -2681.915} C_VEL
LIN {X 0,Y 565.957,Z 473.313,A -85,B 0,C 180,E1 -2684.884,E2 -2684.884} C_VEL
LIN {X 0,Y 565.907,Z 479.213,A -85,B 0,C 180,E1 -2687.402,E2 -2687.402} C_VEL
LIN {X 0,Y 566.92,Z 486.953,A -85,B 0,C 180,E1 -2687.584,E2 -2687.584} C_VEL
LIN {X 0,Y 566.779,Z 499.985,A -85,B 0,C 180,E1 -2687.967,E2 -2687.967} C_VEL
LIN {X 0,Y 566.645,Z 512.178,A -85,B 0,C 180,E1 -2688.473,E2 -2688.473} C_VEL
LIN {X 0,Y 566.558,Z 523.775,A -85,B 0,C 180,E1 -2689.11,E2 -2689.11} C_VEL
LIN {X 0,Y 566.406,Z 535.181,A -85,B 0,C 180,E1 -2689.906,E2 -2689.906} C_VEL
LIN {X 0,Y 566.255,Z 544.557,A -85,B 0,C 180,E1 -2690.715,E2 -2690.715} C_VEL
LIN {X 0,Y 566.158,Z 553.116,A -85,B 0,C 180,E1 -2691.613,E2 -2691.613} C_VEL
LIN {X 0,Y 566.064,Z 561.428,A -85,B 0,C 180,E1 -2692.689,E2 -2692.689} C_VEL
LIN {X 0,Y 565.988,Z 568.124,A -85,B 0,C 180,E1 -2693.763,E2 -2693.763} C_VEL
LIN {X 0,Y 565.878,Z 574.265,A -85,B 0,C 180,E1 -2695.013,E2 -2695.013} C_VEL
LIN {X 0,Y 565.927,Z 578.254,A -85,B 0,C 180,E1 -2696.084,E2 -2696.084} C_VEL
LIN {X 0,Y 565.878,Z 581.202,A -85,B 0,C 180,E1 -2697.153,E2 -2697.153} C_VEL
LIN {X 0,Y 565.839,Z 582.628,A -85,B 0,C 180,E1 -2697.865,E2 -2697.865} C_VEL
LIN {X 0,Y 565.841,Z 584.256,A -85,B 0,C 180,E1 -2699.288,E2 -2699.288} C_VEL
LIN {X 0,Y 565.839,Z 584.496,A -85,B 0,C 180,E1 -2700,E2 -2700} C_VEL
LIN {X 0,Y 565.841,Z 584.314,A -85,B 0,C 180,E1 -2700.712,E2 -2700.712} C_VEL
LIN {X 0,Y 565.838,Z 582.769,A -85,B 0,C 180,E1 -2702.135,E2 -2702.135} C_VEL
LIN {X 0,Y 565.879,Z 581.408,A -85,B 0,C 180,E1 -2702.848,E2 -2702.848} C_VEL
LIN {X 0,Y 565.927,Z 578.53,A -85,B 0,C 180,E1 -2703.917,E2 -2703.917} C_VEL
LIN {X 0,Y 565.878,Z 574.629,A -85,B 0,C 180,E1 -2704.988,E2 -2704.988} C_VEL
LIN {X 0,Y 565.988,Z 569.596,A -85,B 0,C 180,E1 -2706.059,E2 -2706.059} C_VEL
LIN {X 0,Y 566.032,Z 563.271,A -85,B 0,C 180,E1 -2707.132,E2 -2707.132} C_VEL
LIN {X 0,Y 566.129,Z 555.35,A -85,B 0,C 180,E1 -2708.208,E2 -2708.208} C_VEL
LIN {X 0,Y 566.249,Z 545.498,A -85,B 0,C 180,E1 -2709.285,E2 -2709.285} C_VEL
LIN {X 0,Y 566.413,Z 535.176,A -85,B 0,C 180,E1 -2710.184,E2 -2710.184} C_VEL
LIN {X 0,Y 566.526,Z 523.894,A -85,B 0,C 180,E1 -2710.973,E2 -2710.973} C_VEL
LIN {X 0,Y 566.661,Z 512.686,A -85,B 0,C 180,E1 -2711.593,E2 -2711.593} C_VEL
LIN {X 0,Y 566.786,Z 500.09,A -85,B 0,C 180,E1 -2712.119,E2 -2712.119} C_VEL
LIN {X 0,Y 566.916,Z 486.915,A -85,B 0,C 180,E1 -2712.507,E2 -2712.507} C_VEL
LIN {X 0,Y 565.916,Z 479.21,A -85,B 0,C 180,E1 -2712.689,E2 -2712.689} C_VEL
LIN {X 0,Y 565.957,Z 473.523,A -85,B 0,C 180,E1 -2715.116,E2 -2715.116} C_VEL
LIN {X 0,Y 565.99,Z 466.655,A -85,B 0,C 180,E1 -2718.085,E2 -2718.085} C_VEL
LIN {X 0,Y 566.041,Z 459.786,A -85,B 0,C 180,E1 -2721.104,E2 -2721.104} C_VEL
LIN {X 0,Y 566.017,Z 457.48,A -85,B 0,C 180,E1 -2722.133,E2 -2722.133} C_VEL
LIN {X 0,Y 565.351,Z 456.26,A -85,B 0,C 180,E1 -2722.714,E2 -2722.714} C_VEL
LIN {X 0,Y 562.512,Z 454.494,A -85,B 0,C 180,E1 -2723.661,E2 -2723.661} C_VEL
LIN {X 0,Y 560.121,Z 453.107,A -85,B 0,C 180,E1 -2724.424,E2 -2724.424} C_VEL
LIN {X 0,Y 559.105,Z 451.954,A -85,B 0,C 180,E1 -2725.011,E2 -2725.011} C_VEL
LIN {X 0,Y 559.027,Z 451.532,A -85,B 0,C 180,E1 -2725.208,E2 -2725.208} C_VEL
LIN {X 0,Y 559.103,Z 444.784,A -85,B 0,C 180,E1 -2728.368,E2 -2728.368} C_VEL
LIN {X 0,Y 559.164,Z 438.722,A -85,B 0,C 180,E1 -2731.275,E2 -2731.275} C_VEL
LIN {X 0,Y 559.239,Z 433.225,A -85,B 0,C 180,E1 -2733.959,E2 -2733.959} C_VEL
LIN {X 0,Y 559.217,Z 429.456,A -85,B 0,C 180,E1 -2735.871,E2 -2735.871} C_VEL
LIN {X 0,Y 559.178,Z 429.458,A -85,B 0,C 180,E1 -2738.934,E2 -2738.934} C_VEL
LIN {X 0,Y 559.183,Z 429.457,A -85,B 0,C 180,E1 -2742.137,E2 -2742.137} C_VEL
LIN {X 0,Y 559.146,Z 429.463,A -85,B 0,C 180,E1 -2744.739,E2 -2744.739} C_VEL
LIN {X 0,Y 559.162,Z 429.463,A -85,B 0,C 180,E1 -2747.256,E2 -2747.256} C_VEL
LIN {X 0,Y 559.189,Z 429.458,A -85,B 0,C 180,E1 -2750.134,E2 -2750.134} C_VEL
LIN {X 0,Y 559.228,Z 429.619,A -85,B 0,C 180,E1 -2751.875,E2 -2751.875} C_VEL
LIN {X 0,Y 559.308,Z 436.437,A -85,B 0,C 180,E1 -2754.246,E2 -2754.246} C_VEL
LIN {X 0,Y 559.229,Z 444.876,A -85,B 0,C 180,E1 -2757.289,E2 -2757.289} C_VEL
LIN {X 0,Y 559.236,Z 452.755,A -85,B 0,C 180,E1 -2760.128,E2 -2760.128} C_VEL
LIN {X 0,Y 559.236,Z 461.303,A -85,B 0,C 180,E1 -2763.16,E2 -2763.16} C_VEL
LIN {X 0,Y 559.198,Z 468.984,A -85,B 0,C 180,E1 -2765.891,E2 -2765.891} C_VEL
LIN {X 0,Y 559.1,Z 477.534,A -85,B 0,C 180,E1 -2769.006,E2 -2769.006} C_VEL
LIN {X 0,Y 559.016,Z 485.016,A -85,B 0,C 180,E1 -2771.681,E2 -2771.681} C_VEL
LIN {X 0,Y 558.956,Z 493.166,A -85,B 0,C 180,E1 -2774.549,E2 -2774.549} C_VEL
LIN {X 0,Y 560.58,Z 501.851,A -85,B 0,C 180,E1 -2774.748,E2 -2774.748} C_VEL
LIN {X 0,Y 560.405,Z 516.621,A -85,B 0,C 180,E1 -2775.123,E2 -2775.123} C_VEL
LIN {X 0,Y 560.234,Z 528.769,A -85,B 0,C 180,E1 -2775.562,E2 -2775.562} C_VEL
LIN {X 0,Y 560.077,Z 540.715,A -85,B 0,C 180,E1 -2776.113,E2 -2776.113} C_VEL
LIN {X 0,Y 559.823,Z 553.424,A -85,B 0,C 180,E1 -2776.847,E2 -2776.847} C_VEL
LIN {X 0,Y 559.584,Z 566.044,A -85,B 0,C 180,E1 -2777.763,E2 -2777.763} C_VEL
LIN {X 0,Y 559.384,Z 576.232,A -85,B 0,C 180,E1 -2778.665,E2 -2778.665} C_VEL
LIN {X 0,Y 559.312,Z 584.259,A -85,B 0,C 180,E1 -2779.501,E2 -2779.501} C_VEL
LIN {X 0,Y 559.125,Z 593.21,A -85,B 0,C 180,E1 -2780.595,E2 -2780.595} C_VEL
LIN {X 0,Y 558.995,Z 601.775,A -85,B 0,C 180,E1 -2781.868,E2 -2781.868} C_VEL
LIN {X 0,Y 558.904,Z 608.627,A -85,B 0,C 180,E1 -2783.139,E2 -2783.139} C_VEL
LIN {X 0,Y 558.913,Z 613.383,A -85,B 0,C 180,E1 -2784.226,E2 -2784.226} C_VEL
LIN {X 0,Y 558.82,Z 617.212,A -85,B 0,C 180,E1 -2785.31,E2 -2785.31} C_VEL
LIN {X 0,Y 558.826,Z 620.203,A -85,B 0,C 180,E1 -2786.394,E2 -2786.394} C_VEL
LIN {X 0,Y 558.796,Z 621.75,A -85,B 0,C 180,E1 -2787.115,E2 -2787.115} C_VEL
LIN {X 0,Y 558.743,Z 623.784,A -85,B 0,C 180,E1 -2788.558,E2 -2788.558} C_VEL
LIN {X 0,Y 558.739,Z 624.455,A -85,B 0,C 180,E1 -2789.999,E2 -2789.999} C_VEL
LIN {X 0,Y 558.738,Z 624.351,A -85,B 0,C 180,E1 -2790.72,E2 -2790.72} C_VEL
LIN {X 0,Y 558.744,Z 623.034,A -85,B 0,C 180,E1 -2792.162,E2 -2792.162} C_VEL
LIN {X 0,Y 558.794,Z 621.932,A -85,B 0,C 180,E1 -2792.883,E2 -2792.883} C_VEL
LIN {X 0,Y 558.867,Z 618.561,A -85,B 0,C 180,E1 -2794.326,E2 -2794.326} C_VEL
LIN {X 0,Y 558.859,Z 615.106,A -85,B 0,C 180,E1 -2795.411,E2 -2795.411} C_VEL
LIN {X 0,Y 558.894,Z 610.359,A -85,B 0,C 180,E1 -2796.579,E2 -2796.579} C_VEL
LIN {X 0,Y 558.963,Z 604.347,A -85,B 0,C 180,E1 -2797.767,E2 -2797.767} C_VEL
LIN {X 0,Y 559.077,Z 597.699,A -85,B 0,C 180,E1 -2798.857,E2 -2798.857} C_VEL
LIN {X 0,Y 559.185,Z 588.247,A -85,B 0,C 180,E1 -2800.133,E2 -2800.133} C_VEL
LIN {X 0,Y 559.388,Z 578.166,A -85,B 0,C 180,E1 -2801.237,E2 -2801.237} C_VEL
LIN {X 0,Y 559.558,Z 568.232,A -85,B 0,C 180,E1 -2802.143,E2 -2802.143} C_VEL
LIN {X 0,Y 559.75,Z 557.446,A -85,B 0,C 180,E1 -2802.968,E2 -2802.968} C_VEL
LIN {X 0,Y 559.956,Z 545.861,A -85,B 0,C 180,E1 -2803.703,E2 -2803.703} C_VEL
LIN {X 0,Y 560.191,Z 532.066,A -85,B 0,C 180,E1 -2804.391,E2 -2804.391} C_VEL
LIN {X 0,Y 560.353,Z 519.028,A -85,B 0,C 180,E1 -2804.888,E2 -2804.888} C_VEL
LIN {X 0,Y 560.536,Z 505.979,A -85,B 0,C 180,E1 -2805.251,E2 -2805.251} C_VEL
LIN {X 0,Y 560.274,Z 499.823,A -85,B 0,C 180,E1 -2805.386,E2 -2805.386} C_VEL
LIN {X 0,Y 558.941,Z 493.162,A -85,B 0,C 180,E1 -2805.543,E2 -2805.543} C_VEL
LIN {X 0,Y 559.013,Z 485.275,A -85,B 0,C 180,E1 -2808.318,E2 -2808.318} C_VEL
LIN {X 0,Y 559.095,Z 477.789,A -85,B 0,C 180,E1 -2810.992,E2 -2810.992} C_VEL
LIN {X 0,Y 559.195,Z 469.233,A -85,B 0,C 180,E1 -2814.107,E2 -2814.107} C_VEL
LIN {X 0,Y 559.229,Z 461.396,A -85,B 0,C 180,E1 -2816.898,E2 -2816.898} C_VEL
LIN {X 0,Y 559.281,Z 453.018,A -85,B 0,C 180,E1 -2819.881,E2 -2819.881} C_VEL
LIN {X 0,Y 559.287,Z 443.96,A -85,B 0,C 180,E1 -2823.134,E2 -2823.134} C_VEL
LIN {X 0,Y 559.301,Z 436.699,A -85,B 0,C 180,E1 -2825.752,E2 -2825.752} C_VEL
LIN {X 0,Y 559.314,Z 430.235,A -85,B 0,C 180,E1 -2828.001,E2 -2828.001} C_VEL
LIN {X 0,Y 559.21,Z 429.454,A -85,B 0,C 180,E1 -2828.353,E2 -2828.353} C_VEL
LIN {X 0,Y 559.186,Z 429.459,A -85,B 0,C 180,E1 -2831.053,E2 -2831.053} C_VEL
LIN {X 0,Y 559.157,Z 429.457,A -85,B 0,C 180,E1 -2833.731,E2 -2833.731} C_VEL
LIN {X 0,Y 559.167,Z 429.456,A -85,B 0,C 180,E1 -2836.799,E2 -2836.799} C_VEL
LIN {X 0,Y 559.17,Z 429.457,A -85,B 0,C 180,E1 -2839.189,E2 -2839.189} C_VEL
LIN {X 0,Y 559.128,Z 429.46,A -85,B 0,C 180,E1 -2841.982,E2 -2841.982} C_VEL
LIN {X 0,Y 559.152,Z 429.463,A -85,B 0,C 180,E1 -2844.782,E2 -2844.782} C_VEL
LIN {X 0,Y 559.167,Z 429.455,A -85,B 0,C 180,E1 -2847.36,E2 -2847.36} C_VEL
LIN {X 0,Y 559.181,Z 429.459,A -85,B 0,C 180,E1 -2850.134,E2 -2850.134} C_VEL
LIN {X 0,Y 559.173,Z 429.457,A -85,B 0,C 180,E1 -2853.169,E2 -2853.169} C_VEL
LIN {X 0,Y 559.151,Z 429.46,A -85,B 0,C 180,E1 -2855.495,E2 -2855.495} C_VEL
LIN {X 0,Y 559.156,Z 429.459,A -85,B 0,C 180,E1 -2858.447,E2 -2858.447} C_VEL
LIN {X 0,Y 559.163,Z 429.456,A -85,B 0,C 180,E1 -2860.926,E2 -2860.926} C_VEL
LIN {X 0,Y 559.164,Z 429.461,A -85,B 0,C 180,E1 -2863.948,E2 -2863.948} C_VEL
LIN {X 0,Y 559.165,Z 429.456,A -85,B 0,C 180,E1 -2866.184,E2 -2866.184} C_VEL
LIN {X 0,Y 559.224,Z 429.454,A -85,B 0,C 180,E1 -2869.134,E2 -2869.134} C_VEL
LIN {X 0,Y 559.204,Z 429.451,A -85,B 0,C 180,E1 -2872.054,E2 -2872.054} C_VEL
LIN {X 0,Y 559.252,Z 429.443,A -85,B 0,C 180,E1 -2874.953,E2 -2874.953} C_VEL
LIN {X 0,Y 559.243,Z 429.45,A -85,B 0,C 180,E1 -2877.839,E2 -2877.839} C_VEL
LIN {X 0,Y 559.267,Z 429.444,A -85,B 0,C 180,E1 -2880.72,E2 -2880.72} C_VEL
LIN {X 0,Y 559.238,Z 429.449,A -85,B 0,C 180,E1 -2882.881,E2 -2882.881} C_VEL
LIN {X 0,Y 559.223,Z 429.447,A -85,B 0,C 180,E1 -2885.77,E2 -2885.77} C_VEL
LIN {X 0,Y 559.196,Z 429.451,A -85,B 0,C 180,E1 -2888.674,E2 -2888.674} C_VEL
LIN {X 0,Y 559.199,Z 429.455,A -85,B 0,C 180,E1 -2891.601,E2 -2891.601} C_VEL
LIN {X 0,Y 559.188,Z 429.454,A -85,B 0,C 180,E1 -2894.596,E2 -2894.596} C_VEL
LIN {X 0,Y 559.155,Z 429.452,A -85,B 0,C 180,E1 -2897.557,E2 -2897.557} C_VEL
LIN {X 0,Y 559.166,Z 429.457,A -85,B 0,C 180,E1 -2899.838,E2 -2899.838} C_VEL
LIN {X 0,Y 559.135,Z 429.463,A -85,B 0,C 180,E1 -2902.153,E2 -2902.153} C_VEL
LIN {X 0,Y 559.17,Z 429.458,A -85,B 0,C 180,E1 -2905.188,E2 -2905.188} C_VEL
LIN {X 0,Y 559.186,Z 429.453,A -85,B 0,C 180,E1 -2907.712,E2 -2907.712} C_VEL
LIN {X 0,Y 559.161,Z 429.458,A -85,B 0,C 180,E1 -2910.182,E2 -2910.182} C_VEL
LIN {X 0,Y 559.168,Z 429.457,A -85,B 0,C 180,E1 -2912.715,E2 -2912.715} C_VEL
LIN {X 0,Y 559.15,Z 429.458,A -85,B 0,C 180,E1 -2915.322,E2 -2915.322} C_VEL
LIN {X 0,Y 559.127,Z 429.461,A -85,B 0,C 180,E1 -2918.018,E2 -2918.018} C_VEL
LIN {X 0,Y 559.173,Z 429.459,A -85,B 0,C 180,E1 -2920.811,E2 -2920.811} C_VEL
LIN {X 0,Y 559.158,Z 429.456,A -85,B 0,C 180,E1 -2923.732,E2 -2923.732} C_VEL
LIN {X 0,Y 559.14,Z 429.459,A -85,B 0,C 180,E1 -2926.804,E2 -2926.804} C_VEL
LIN {X 0,Y 559.171,Z 429.457,A -85,B 0,C 180,E1 -2929.191,E2 -2929.191} C_VEL
LIN {X 0,Y 559.13,Z 429.461,A -85,B 0,C 180,E1 -2931.984,E2 -2931.984} C_VEL
LIN {X 0,Y 559.157,Z 429.463,A -85,B 0,C 180,E1 -2934.784,E2 -2934.784} C_VEL
LIN {X 0,Y 559.201,Z 429.633,A -85,B 0,C 180,E1 -2936.189,E2 -2936.189} C_VEL
LIN {X 0,Y 560.101,Z 435.024,A -85,B 0,C 180,E1 -2937.774,E2 -2937.774} C_VEL
LIN {X 0,Y 559.927,Z 444.518,A -85,B 0,C 180,E1 -2940.346,E2 -2940.346} C_VEL
LIN {X 0,Y 559.716,Z 455.161,A -85,B 0,C 180,E1 -2943.127,E2 -2943.127} C_VEL
LIN {X 0,Y 559.535,Z 466.062,A -85,B 0,C 180,E1 -2945.909,E2 -2945.909} C_VEL
LIN {X 0,Y 559.347,Z 478.55,A -85,B 0,C 180,E1 -2949.018,E2 -2949.018} C_VEL
LIN {X 0,Y 559.223,Z 491.039,A -85,B 0,C 180,E1 -2952.068,E2 -2952.068} C_VEL
LIN {X 0,Y 559.126,Z 501.089,A -85,B 0,C 180,E1 -2954.486,E2 -2954.486} C_VEL
LIN {X 0,Y 560.572,Z 508.701,A -85,B 0,C 180,E1 -2954.643,E2 -2954.643} C_VEL
LIN {X 0,Y 560.457,Z 522.794,A -85,B 0,C 180,E1 -2954.963,E2 -2954.963} C_VEL
LIN {X 0,Y 560.294,Z 536.512,A -85,B 0,C 180,E1 -2955.422,E2 -2955.422} C_VEL
LIN {X 0,Y 560.106,Z 549.898,A -85,B 0,C 180,E1 -2956.024,E2 -2956.024} C_VEL
LIN {X 0,Y 559.805,Z 562.696,A -85,B 0,C 180,E1 -2956.756,E2 -2956.756} C_VEL
LIN {X 0,Y 559.645,Z 574.327,A -85,B 0,C 180,E1 -2957.582,E2 -2957.582} C_VEL
LIN {X 0,Y 559.389,Z 585.152,A -85,B 0,C 180,E1 -2958.513,E2 -2958.513} C_VEL
LIN {X 0,Y 559.272,Z 594.716,A -85,B 0,C 180,E1 -2959.502,E2 -2959.502} C_VEL
LIN {X 0,Y 559.12,Z 603.566,A -85,B 0,C 180,E1 -2960.596,E2 -2960.596} C_VEL
LIN {X 0,Y 558.985,Z 612.042,A -85,B 0,C 180,E1 -2961.87,E2 -2961.87} C_VEL
LIN {X 0,Y 558.901,Z 618.871,A -85,B 0,C 180,E1 -2963.14,E2 -2963.14} C_VEL
LIN {X 0,Y 558.912,Z 623.572,A -85,B 0,C 180,E1 -2964.228,E2 -2964.228} C_VEL
LIN {X 0,Y 558.865,Z 628.446,A -85,B 0,C 180,E1 -2965.674,E2 -2965.674} C_VEL
LIN {X 0,Y 558.795,Z 631.833,A -85,B 0,C 180,E1 -2967.117,E2 -2967.117} C_VEL
LIN {X 0,Y 558.74,Z 633.834,A -85,B 0,C 180,E1 -2968.559,E2 -2968.559} C_VEL
LIN {X 0,Y 558.738,Z 634.5,A -85,B 0,C 180,E1 -2970.001,E2 -2970.001} C_VEL
LIN {X 0,Y 558.74,Z 633.833,A -85,B 0,C 180,E1 -2971.442,E2 -2971.442} C_VEL
LIN {X 0,Y 558.796,Z 631.832,A -85,B 0,C 180,E1 -2972.885,E2 -2972.885} C_VEL
LIN {X 0,Y 558.865,Z 628.443,A -85,B 0,C 180,E1 -2974.328,E2 -2974.328} C_VEL
LIN {X 0,Y 558.911,Z 623.565,A -85,B 0,C 180,E1 -2975.774,E2 -2975.774} C_VEL
LIN {X 0,Y 558.903,Z 618.861,A -85,B 0,C 180,E1 -2976.861,E2 -2976.861} C_VEL
LIN {X 0,Y 558.987,Z 612.032,A -85,B 0,C 180,E1 -2978.132,E2 -2978.132} C_VEL
LIN {X 0,Y 559.118,Z 603.552,A -85,B 0,C 180,E1 -2979.406,E2 -2979.406} C_VEL
LIN {X 0,Y 559.273,Z 594.7,A -85,B 0,C 180,E1 -2980.499,E2 -2980.499} C_VEL
LIN {X 0,Y 559.489,Z 583.981,A -85,B 0,C 180,E1 -2981.595,E2 -2981.595} C_VEL
LIN {X 0,Y 559.647,Z 573.13,A -85,B 0,C 180,E1 -2982.512,E2 -2982.512} C_VEL
LIN {X 0,Y 559.852,Z 561.244,A -85,B 0,C 180,E1 -2983.337,E2 -2983.337} C_VEL
LIN {X 0,Y 560.152,Z 548.079,A -85,B 0,C 180,E1 -2984.07,E2 -2984.07} C_VEL
LIN {X 0,Y 560.33,Z 535.233,A -85,B 0,C 180,E1 -2984.628,E2 -2984.628} C_VEL
LIN {X 0,Y 560.488,Z 521.372,A -85,B 0,C 180,E1 -2985.074,E2 -2985.074} C_VEL
LIN {X 0,Y 560.448,Z 508.038,A -85,B 0,C 180,E1 -2985.371,E2 -2985.371} C_VEL
LIN {X 0,Y 559.107,Z 501.081,A -85,B 0,C 180,E1 -2985.517,E2 -2985.517} C_VEL
LIN {X 0,Y 559.258,Z 489.47,A -85,B 0,C 180,E1 -2988.311,E2 -2988.311} C_VEL
LIN {X 0,Y 559.375,Z 476.982,A -85,B 0,C 180,E1 -2991.369,E2 -2991.369} C_VEL
LIN {X 0,Y 559.541,Z 466.054,A -85,B 0,C 180,E1 -2994.093,E2 -2994.093} C_VEL
LIN {X 0,Y 559.702,Z 454.739,A -85,B 0,C 180,E1 -2996.934,E2 -2996.934} C_VEL
LIN {X 0,Y 560.035,Z 442.879,A -85,B 0,C 180,E1 -3000.131,E2 -3000.131} C_VEL
LIN {X 0,Y 560.238,Z 435.661,A -85,B 0,C 180,E1 -3002.219,E2 -3002.219} C_VEL
LIN {X 0,Y 559.203,Z 429.457,A -85,B 0,C 180,E1 -3004.321,E2 -3004.321} C_VEL
LIN {X 0,Y 559.148,Z 429.462,A -85,B 0,C 180,E1 -3007.109,E2 -3007.109} C_VEL
LIN {X 0,Y 559.169,Z 429.459,A -85,B 0,C 180,E1 -3009.943,E2 -3009.943} C_VEL
LIN {X 0,Y 559.162,Z 429.459,A -85,B 0,C 180,E1 -3012.744,E2 -3012.744} C_VEL
LIN {X 0,Y 559.159,Z 429.46,A -85,B 0,C 180,E1 -3015.761,E2 -3015.761} C_VEL
LIN {X 0,Y 559.189,Z 429.457,A -85,B 0,C 180,E1 -3018.232,E2 -3018.232} C_VEL
LIN {X 0,Y 559.177,Z 429.459,A -85,B 0,C 180,E1 -3021.192,E2 -3021.192} C_VEL
LIN {X 0,Y 559.195,Z 429.534,A -85,B 0,C 180,E1 -3024.238,E2 -3024.238} C_VEL
LIN {X 0,Y 559.306,Z 432.197,A -85,B 0,C 180,E1 -3025.566,E2 -3025.566} C_VEL
LIN {X 0,Y 559.187,Z 438.696,A -85,B 0,C 180,E1 -3028.721,E2 -3028.721} C_VEL
LIN {X 0,Y 559.137,Z 444.774,A -85,B 0,C 180,E1 -3031.626,E2 -3031.626} C_VEL
LIN {X 0,Y 559.079,Z 449.697,A -85,B 0,C 180,E1 -3033.898,E2 -3033.898} C_VEL
LIN {X 0,Y 559.007,Z 455.301,A -85,B 0,C 180,E1 -3036.604,E2 -3036.604} C_VEL
LIN {X 0,Y 558.931,Z 461.302,A -85,B 0,C 180,E1 -3039.386,E2 -3039.386} C_VEL
LIN {X 0,Y 558.911,Z 468.166,A -85,B 0,C 180,E1 -3042.435,E2 -3042.435} C_VEL
LIN {X 0,Y 558.871,Z 475.27,A -85,B 0,C 180,E1 -3045.537,E2 -3045.537} C_VEL
LIN {X 0,Y 558.844,Z 479.214,A -85,B 0,C 180,E1 -3047.24,E2 -3047.24} C_VEL
LIN {X 0,Y 559.982,Z 486.975,A -85,B 0,C 180,E1 -3047.428,E2 -3047.428} C_VEL
LIN {X 0,Y 559.847,Z 500.002,A -85,B 0,C 180,E1 -3047.816,E2 -3047.816} C_VEL
LIN {X 0,Y 559.688,Z 512.191,A -85,B 0,C 180,E1 -3048.327,E2 -3048.327} C_VEL
LIN {X 0,Y 559.583,Z 523.93,A -85,B 0,C 180,E1 -3048.982,E2 -3048.982} C_VEL
LIN {X 0,Y 559.415,Z 535.19,A -85,B 0,C 180,E1 -3049.779,E2 -3049.779} C_VEL
LIN {X 0,Y 559.239,Z 544.564,A -85,B 0,C 180,E1 -3050.597,E2 -3050.597} C_VEL
LIN {X 0,Y 559.129,Z 553.121,A -85,B 0,C 180,E1 -3051.507,E2 -3051.507} C_VEL
LIN {X 0,Y 558.989,Z 561.432,A -85,B 0,C 180,E1 -3052.596,E2 -3052.596} C_VEL
LIN {X 0,Y 558.89,Z 567.918,A -85,B 0,C 180,E1 -3053.645,E2 -3053.645} C_VEL
LIN {X 0,Y 558.869,Z 572.665,A -85,B 0,C 180,E1 -3054.588,E2 -3054.588} C_VEL
LIN {X 0,Y 558.869,Z 577.023,A -85,B 0,C 180,E1 -3055.673,E2 -3055.673} C_VEL
LIN {X 0,Y 558.837,Z 579.328,A -85,B 0,C 180,E1 -3056.395,E2 -3056.395} C_VEL
LIN {X 0,Y 558.8,Z 581.204,A -85,B 0,C 180,E1 -3057.116,E2 -3057.116} C_VEL
LIN {X 0,Y 558.745,Z 582.629,A -85,B 0,C 180,E1 -3057.838,E2 -3057.838} C_VEL
LIN {X 0,Y 558.742,Z 584.256,A -85,B 0,C 180,E1 -3059.279,E2 -3059.279} C_VEL
LIN {X 0,Y 558.74,Z 584.496,A -85,B 0,C 180,E1 -3060,E2 -3060} C_VEL
LIN {X 0,Y 558.741,Z 584.314,A -85,B 0,C 180,E1 -3060.721,E2 -3060.721} C_VEL
LIN {X 0,Y 558.745,Z 582.767,A -85,B 0,C 180,E1 -3062.163,E2 -3062.163} C_VEL
LIN {X 0,Y 558.8,Z 581.406,A -85,B 0,C 180,E1 -3062.884,E2 -3062.884} C_VEL
LIN {X 0,Y 558.844,Z 578.528,A -85,B 0,C 180,E1 -3063.966,E2 -3063.966} C_VEL
LIN {X 0,Y 558.798,Z 574.627,A -85,B 0,C 180,E1 -3065.051,E2 -3065.051} C_VEL
LIN {X 0,Y 558.908,Z 569.594,A -85,B 0,C 180,E1 -3066.136,E2 -3066.136} C_VEL
LIN {X 0,Y 558.973,Z 563.268,A -85,B 0,C 180,E1 -3067.223,E2 -3067.223} C_VEL
LIN {X 0,Y 559.091,Z 555.345,A -85,B 0,C 180,E1 -3068.312,E2 -3068.312} C_VEL
LIN {X 0,Y 559.224,Z 545.492,A -85,B 0,C 180,E1 -3069.403,E2 -3069.403} C_VEL
LIN {X 0,Y 559.399,Z 535.17,A -85,B 0,C 180,E1 -3070.313,E2 -3070.313} C_VEL
LIN {X 0,Y 559.539,Z 524.143,A -85,B 0,C 180,E1 -3071.095,E2 -3071.095} C_VEL
LIN {X 0,Y 559.693,Z 512.674,A -85,B 0,C 180,E1 -3071.739,E2 -3071.739} C_VEL
LIN {X 0,Y 559.854,Z 500.075,A -85,B 0,C 180,E1 -3072.271,E2 -3072.271} C_VEL
LIN {X 0,Y 559.999,Z 486.891,A -85,B 0,C 180,E1 -3072.664,E2 -3072.664} C_VEL
LIN {X 0,Y 558.821,Z 479.209,A -85,B 0,C 180,E1 -3072.853,E2 -3072.853} C_VEL
LIN {X 0,Y 558.868,Z 473.521,A -85,B 0,C 180,E1 -3075.313,E2 -3075.313} C_VEL
LIN {X 0,Y 558.906,Z 466.653,A -85,B 0,C 180,E1 -3078.323,E2 -3078.323} C_VEL
LIN {X 0,Y 558.997,Z 459.51,A -85,B 0,C 180,E1 -3081.507,E2 -3081.507} C_VEL
LIN {X 0,Y 558.999,Z 453.027,A -85,B 0,C 180,E1 -3084.513,E2 -3084.513} C_VEL
LIN {X 0,Y 559.027,Z 451.532,A -85,B 0,C 180,E1 -3085.208,E2 -3085.208} C_VEL
LIN {X 0,Y 558.368,Z 450.332,A -85,B 0,C 180,E1 -3085.797,E2 -3085.797} C_VEL
LIN {X 0,Y 555.506,Z 448.607,A -85,B 0,C 180,E1 -3086.759,E2 -3086.759} C_VEL
LIN {X 0,Y 553.107,Z 447.262,A -85,B 0,C 180,E1 -3087.533,E2 -3087.533} C_VEL
LIN {X 0,Y 552.111,Z 446.13,A -85,B 0,C 180,E1 -3088.129,E2 -3088.129} C_VEL
LIN {X 0,Y 552.048,Z 445.718,A -85,B 0,C 180,E1 -3088.329,E2 -3088.329} C_VEL
LIN {X 0,Y 552.086,Z 441.007,A -85,B 0,C 180,E1 -3090.61,E2 -3090.61} C_VEL
LIN {X 0,Y 552.187,Z 435.764,A -85,B 0,C 180,E1 -3093.181,E2 -3093.181} C_VEL
LIN {X 0,Y 552.154,Z 430.335,A -85,B 0,C 180,E1 -3095.951,E2 -3095.951} C_VEL
LIN {X 0,Y 552.125,Z 430.337,A -85,B 0,C 180,E1 -3099.061,E2 -3099.061} C_VEL
LIN {X 0,Y 552.138,Z 430.336,A -85,B 0,C 180,E1 -3101.445,E2 -3101.445} C_VEL
LIN {X 0,Y 552.103,Z 430.339,A -85,B 0,C 180,E1 -3104.532,E2 -3104.532} C_VEL
LIN {X 0,Y 552.135,Z 430.337,A -85,B 0,C 180,E1 -3107.584,E2 -3107.584} C_VEL
LIN {X 0,Y 552.14,Z 430.338,A -85,B 0,C 180,E1 -3110.473,E2 -3110.473} C_VEL
LIN {X 0,Y 552.192,Z 430.445,A -85,B 0,C 180,E1 -3111.785,E2 -3111.785} C_VEL
LIN {X 0,Y 552.277,Z 437.26,A -85,B 0,C 180,E1 -3114.17,E2 -3114.17} C_VEL
LIN {X 0,Y 552.221,Z 445.426,A -85,B 0,C 180,E1 -3117.137,E2 -3117.137} C_VEL
LIN {X 0,Y 552.2,Z 453.102,A -85,B 0,C 180,E1 -3119.935,E2 -3119.935} C_VEL
LIN {X 0,Y 552.189,Z 461.616,A -85,B 0,C 180,E1 -3122.99,E2 -3122.99} C_VEL
LIN {X 0,Y 552.125,Z 469.908,A -85,B 0,C 180,E1 -3125.962,E2 -3125.962} C_VEL
LIN {X 0,Y 552.053,Z 477.536,A -85,B 0,C 180,E1 -3128.725,E2 -3128.725} C_VEL
LIN {X 0,Y 551.948,Z 485.018,A -85,B 0,C 180,E1 -3131.437,E2 -3131.437} C_VEL
LIN {X 0,Y 551.875,Z 493.168,A -85,B 0,C 180,E1 -3134.346,E2 -3134.346} C_VEL
LIN {X 0,Y 553.722,Z 502.655,A -85,B 0,C 180,E1 -3134.571,E2 -3134.571} C_VEL
LIN {X 0,Y 553.549,Z 517.138,A -85,B 0,C 180,E1 -3134.952,E2 -3134.952} C_VEL
LIN {X 0,Y 553.323,Z 528.769,A -85,B 0,C 180,E1 -3135.377,E2 -3135.377} C_VEL
LIN {X 0,Y 553.179,Z 540.712,A -85,B 0,C 180,E1 -3135.937,E2 -3135.937} C_VEL
LIN {X 0,Y 552.885,Z 553.438,A -85,B 0,C 180,E1 -3136.679,E2 -3136.679} C_VEL
LIN {X 0,Y 552.62,Z 566.04,A -85,B 0,C 180,E1 -3137.607,E2 -3137.607} C_VEL
LIN {X 0,Y 552.407,Z 576.229,A -85,B 0,C 180,E1 -3138.52,E2 -3138.52} C_VEL
LIN {X 0,Y 552.291,Z 584.258,A -85,B 0,C 180,E1 -3139.366,E2 -3139.366} C_VEL
LIN {X 0,Y 552.116,Z 591.812,A -85,B 0,C 180,E1 -3140.289,E2 -3140.289} C_VEL
LIN {X 0,Y 551.964,Z 599.479,A -85,B 0,C 180,E1 -3141.395,E2 -3141.395} C_VEL
LIN {X 0,Y 551.835,Z 606.845,A -85,B 0,C 180,E1 -3142.682,E2 -3142.682} C_VEL
LIN {X 0,Y 551.821,Z 613.38,A -85,B 0,C 180,E1 -3144.151,E2 -3144.151} C_VEL
LIN {X 0,Y 551.717,Z 617.209,A -85,B 0,C 180,E1 -3145.25,E2 -3145.25} C_VEL
LIN {X 0,Y 551.741,Z 620.198,A -85,B 0,C 180,E1 -3146.348,E2 -3146.348} C_VEL
LIN {X 0,Y 551.72,Z 621.753,A -85,B 0,C 180,E1 -3147.078,E2 -3147.078} C_VEL
LIN {X 0,Y 551.643,Z 623.779,A -85,B 0,C 180,E1 -3148.539,E2 -3148.539} C_VEL
LIN {X 0,Y 551.64,Z 624.449,A -85,B 0,C 180,E1 -3149.999,E2 -3149.999} C_VEL
LIN {X 0,Y 551.638,Z 624.349,A -85,B 0,C 180,E1 -3150.729,E2 -3150.729} C_VEL
LIN {X 0,Y 551.655,Z 623.029,A -85,B 0,C 180,E1 -3152.189,E2 -3152.189} C_VEL
LIN {X 0,Y 551.719,Z 621.932,A -85,B 0,C 180,E1 -3152.92,E2 -3152.92} C_VEL
LIN {X 0,Y 551.761,Z 618.557,A -85,B 0,C 180,E1 -3154.382,E2 -3154.382} C_VEL
LIN {X 0,Y 551.789,Z 615.098,A -85,B 0,C 180,E1 -3155.481,E2 -3155.481} C_VEL
LIN {X 0,Y 551.822,Z 610.729,A -85,B 0,C 180,E1 -3156.581,E2 -3156.581} C_VEL
LIN {X 0,Y 551.909,Z 604.339,A -85,B 0,C 180,E1 -3157.867,E2 -3157.867} C_VEL
LIN {X 0,Y 552.006,Z 597.688,A -85,B 0,C 180,E1 -3158.972,E2 -3158.972} C_VEL
LIN {X 0,Y 552.174,Z 588.245,A -85,B 0,C 180,E1 -3160.263,E2 -3160.263} C_VEL
LIN {X 0,Y 552.371,Z 577.8,A -85,B 0,C 180,E1 -3161.416,E2 -3161.416} C_VEL
LIN {X 0,Y 552.577,Z 568.214,A -85,B 0,C 180,E1 -3162.299,E2 -3162.299} C_VEL
LIN {X 0,Y 552.813,Z 557.43,A -85,B 0,C 180,E1 -3163.134,E2 -3163.134} C_VEL
LIN {X 0,Y 553.05,Z 545.852,A -85,B 0,C 180,E1 -3163.877,E2 -3163.877} C_VEL
LIN {X 0,Y 553.314,Z 532.038,A -85,B 0,C 180,E1 -3164.574,E2 -3164.574} C_VEL
LIN {X 0,Y 553.477,Z 519.528,A -85,B 0,C 180,E1 -3165.059,E2 -3165.059} C_VEL
LIN {X 0,Y 553.681,Z 507.023,A -85,B 0,C 180,E1 -3165.417,E2 -3165.417} C_VEL
LIN {X 0,Y 553.485,Z 501.133,A -85,B 0,C 180,E1 -3165.555,E2 -3165.555} C_VEL
LIN {X 0,Y 551.875,Z 493.16,A -85,B 0,C 180,E1 -3165.747,E2 -3165.747} C_VEL
LIN {X 0,Y 551.944,Z 485.273,A -85,B 0,C 180,E1 -3168.561,E2 -3168.561} C_VEL
LIN {X 0,Y 552.047,Z 477.787,A -85,B 0,C 180,E1 -3171.273,E2 -3171.273} C_VEL
LIN {X 0,Y 552.134,Z 469.065,A -85,B 0,C 180,E1 -3174.435,E2 -3174.435} C_VEL
LIN {X 0,Y 552.179,Z 461.153,A -85,B 0,C 180,E1 -3177.27,E2 -3177.27} C_VEL
LIN {X 0,Y 552.22,Z 453.356,A -85,B 0,C 180,E1 -3180.069,E2 -3180.069} C_VEL
LIN {X 0,Y 552.254,Z 444.826,A -85,B 0,C 180,E1 -3183.175,E2 -3183.175} C_VEL
LIN {X 0,Y 552.284,Z 436.271,A -85,B 0,C 180,E1 -3186.27,E2 -3186.27} C_VEL
LIN {X 0,Y 552.185,Z 430.33,A -85,B 0,C 180,E1 -3188.354,E2 -3188.354} C_VEL
LIN {X 0,Y 552.135,Z 430.333,A -85,B 0,C 180,E1 -3191.443,E2 -3191.443} C_VEL
LIN {X 0,Y 552.091,Z 430.342,A -85,B 0,C 180,E1 -3194.531,E2 -3194.531} C_VEL
LIN {X 0,Y 552.125,Z 430.337,A -85,B 0,C 180,E1 -3197.583,E2 -3197.583} C_VEL
LIN {X 0,Y 552.127,Z 430.331,A -85,B 0,C 180,E1 -3200.472,E2 -3200.472} C_VEL
LIN {X 0,Y 552.107,Z 430.338,A -85,B 0,C 180,E1 -3203.315,E2 -3203.315} C_VEL
LIN {X 0,Y 552.132,Z 430.331,A -85,B 0,C 180,E1 -3205.939,E2 -3205.939} C_VEL
LIN {X 0,Y 552.11,Z 430.336,A -85,B 0,C 180,E1 -3208.54,E2 -3208.54} C_VEL
LIN {X 0,Y 552.118,Z 430.337,A -85,B 0,C 180,E1 -3211.437,E2 -3211.437} C_VEL
LIN {X 0,Y 552.128,Z 430.331,A -85,B 0,C 180,E1 -3214.356,E2 -3214.356} C_VEL
LIN {X 0,Y 552.131,Z 430.336,A -85,B 0,C 180,E1 -3216.759,E2 -3216.759} C_VEL
LIN {X 0,Y 552.119,Z 430.334,A -85,B 0,C 180,E1 -3219.12,E2 -3219.12} C_VEL
LIN {X 0,Y 552.124,Z 430.332,A -85,B 0,C 180,E1 -3221.444,E2 -3221.444} C_VEL
LIN {X 0,Y 552.114,Z 430.339,A -85,B 0,C 180,E1 -3223.737,E2 -3223.737} C_VEL
LIN {X 0,Y 552.127,Z 430.334,A -85,B 0,C 180,E1 -3226.004,E2 -3226.004} C_VEL
LIN {X 0,Y 552.184,Z 430.33,A -85,B 0,C 180,E1 -3228.994,E2 -3228.994} C_VEL
LIN {X 0,Y 552.157,Z 430.328,A -85,B 0,C 180,E1 -3231.951,E2 -3231.951} C_VEL
LIN {X 0,Y 552.227,Z 430.319,A -85,B 0,C 180,E1 -3234.889,E2 -3234.889} C_VEL
LIN {X 0,Y 552.214,Z 430.326,A -85,B 0,C 180,E1 -3237.812,E2 -3237.812} C_VEL
LIN {X 0,Y 552.237,Z 430.32,A -85,B 0,C 180,E1 -3240.729,E2 -3240.729} C_VEL
LIN {X 0,Y 552.204,Z 430.324,A -85,B 0,C 180,E1 -3242.918,E2 -3242.918} C_VEL
LIN {X 0,Y 552.193,Z 430.323,A -85,B 0,C 180,E1 -3245.844,E2 -3245.844} C_VEL
LIN {X 0,Y 552.163,Z 430.326,A -85,B 0,C 180,E1 -3248.786,E2 -3248.786} C_VEL
LIN {X 0,Y 552.154,Z 430.332,A -85,B 0,C 180,E1 -3251.751,E2 -3251.751} C_VEL
LIN {X 0,Y 552.127,Z 430.335,A -85,B 0,C 180,E1 -3254.749,E2 -3254.749} C_VEL
LIN {X 0,Y 552.106,Z 430.33,A -85,B 0,C 180,E1 -3257.789,E2 -3257.789} C_VEL
LIN {X 0,Y 552.125,Z 430.337,A -85,B 0,C 180,E1 -3260.101,E2 -3260.101} C_VEL
LIN {X 0,Y 552.089,Z 430.337,A -85,B 0,C 180,E1 -3262.451,E2 -3262.451} C_VEL
LIN {X 0,Y 552.147,Z 430.335,A -85,B 0,C 180,E1 -3265.351,E2 -3265.351} C_VEL
LIN {X 0,Y 552.118,Z 430.332,A -85,B 0,C 180,E1 -3268.098,E2 -3268.098} C_VEL
LIN {X 0,Y 552.106,Z 430.341,A -85,B 0,C 180,E1 -3270.609,E2 -3270.609} C_VEL
LIN {X 0,Y 552.121,Z 430.332,A -85,B 0,C 180,E1 -3273.185,E2 -3273.185} C_VEL
LIN {X 0,Y 552.105,Z 430.341,A -85,B 0,C 180,E1 -3275.842,E2 -3275.842} C_VEL
LIN {X 0,Y 552.118,Z 430.337,A -85,B 0,C 180,E1 -3279.063,E2 -3279.063} C_VEL
LIN {X 0,Y 552.165,Z 430.329,A -85,B 0,C 180,E1 -3281.442,E2 -3281.442} C_VEL
LIN {X 0,Y 552.09,Z 430.343,A -85,B 0,C 180,E1 -3284.533,E2 -3284.533} C_VEL
LIN {X 0,Y 552.124,Z 430.335,A -85,B 0,C 180,E1 -3287.585,E2 -3287.585} C_VEL
LIN {X 0,Y 552.13,Z 430.332,A -85,B 0,C 180,E1 -3290.474,E2 -3290.474} C_VEL
LIN {X 0,Y 552.11,Z 430.339,A -85,B 0,C 180,E1 -3293.317,E2 -3293.317} C_VEL
LIN {X 0,Y 552.156,Z 430.54,A -85,B 0,C 180,E1 -3295.943,E2 -3295.943} C_VEL
LIN {X 0,Y 553.188,Z 436.609,A -85,B 0,C 180,E1 -3297.753,E2 -3297.753} C_VEL
LIN {X 0,Y 552.976,Z 445.845,A -85,B 0,C 180,E1 -3300.288,E2 -3300.288} C_VEL
LIN {X 0,Y 552.742,Z 456.935,A -85,B 0,C 180,E1 -3303.227,E2 -3303.227} C_VEL
LIN {X 0,Y 552.523,Z 467.546,A -85,B 0,C 180,E1 -3305.983,E2 -3305.983} C_VEL
LIN {X 0,Y 552.348,Z 478.55,A -85,B 0,C 180,E1 -3308.739,E2 -3308.739} C_VEL
LIN {X 0,Y 552.203,Z 491.039,A -85,B 0,C 180,E1 -3311.832,E2 -3311.832} C_VEL
LIN {X 0,Y 552.05,Z 501.089,A -85,B 0,C 180,E1 -3314.282,E2 -3314.282} C_VEL
LIN {X 0,Y 553.72,Z 510.221,A -85,B 0,C 180,E1 -3314.478,E2 -3314.478} C_VEL
LIN {X 0,Y 553.558,Z 524.628,A -85,B 0,C 180,E1 -3314.827,E2 -3314.827} C_VEL
LIN {X 0,Y 553.333,Z 538.863,A -85,B 0,C 180,E1 -3315.332,E2 -3315.332} C_VEL
LIN {X 0,Y 553.182,Z 551.661,A -85,B 0,C 180,E1 -3315.939,E2 -3315.939} C_VEL
LIN {X 0,Y 552.865,Z 564.119,A -85,B 0,C 180,E1 -3316.68,E2 -3316.68} C_VEL
LIN {X 0,Y 552.627,Z 576.657,A -85,B 0,C 180,E1 -3317.609,E2 -3317.609} C_VEL
LIN {X 0,Y 552.406,Z 587.514,A -85,B 0,C 180,E1 -3318.594,E2 -3318.594} C_VEL
LIN {X 0,Y 552.178,Z 597.86,A -85,B 0,C 180,E1 -3319.737,E2 -3319.737} C_VEL
LIN {X 0,Y 552.031,Z 606.18,A -85,B 0,C 180,E1 -3320.844,E2 -3320.844} C_VEL
LIN {X 0,Y 551.912,Z 614.133,A -85,B 0,C 180,E1 -3322.133,E2 -3322.133} C_VEL
LIN {X 0,Y 551.821,Z 620.532,A -85,B 0,C 180,E1 -3323.419,E2 -3323.419} C_VEL
LIN {X 0,Y 551.792,Z 624.964,A -85,B 0,C 180,E1 -3324.519,E2 -3324.519} C_VEL
LIN {X 0,Y 551.759,Z 628.446,A -85,B 0,C 180,E1 -3325.618,E2 -3325.618} C_VEL
LIN {X 0,Y 551.719,Z 631.834,A -85,B 0,C 180,E1 -3327.08,E2 -3327.08} C_VEL
LIN {X 0,Y 551.64,Z 633.834,A -85,B 0,C 180,E1 -3328.541,E2 -3328.541} C_VEL
LIN {X 0,Y 551.639,Z 634.5,A -85,B 0,C 180,E1 -3330.001,E2 -3330.001} C_VEL
LIN {X 0,Y 551.64,Z 633.833,A -85,B 0,C 180,E1 -3331.461,E2 -3331.461} C_VEL
LIN {X 0,Y 551.72,Z 631.833,A -85,B 0,C 180,E1 -3332.922,E2 -3332.922} C_VEL
LIN {X 0,Y 551.76,Z 628.443,A -85,B 0,C 180,E1 -3334.384,E2 -3334.384} C_VEL
LIN {X 0,Y 551.818,Z 623.565,A -85,B 0,C 180,E1 -3335.849,E2 -3335.849} C_VEL
LIN {X 0,Y 551.834,Z 617.049,A -85,B 0,C 180,E1 -3337.318,E2 -3337.318} C_VEL
LIN {X 0,Y 551.963,Z 609.796,A -85,B 0,C 180,E1 -3338.605,E2 -3338.605} C_VEL
LIN {X 0,Y 552.116,Z 600.815,A -85,B 0,C 180,E1 -3339.896,E2 -3339.896} C_VEL
LIN {X 0,Y 552.347,Z 591.384,A -85,B 0,C 180,E1 -3341.004,E2 -3341.004} C_VEL
LIN {X 0,Y 552.505,Z 580.943,A -85,B 0,C 180,E1 -3342.023,E2 -3342.023} C_VEL
LIN {X 0,Y 552.768,Z 569.422,A -85,B 0,C 180,E1 -3342.95,E2 -3342.95} C_VEL
LIN {X 0,Y 553.012,Z 556.628,A -85,B 0,C 180,E1 -3343.786,E2 -3343.786} C_VEL
LIN {X 0,Y 553.26,Z 544.133,A -85,B 0,C 180,E1 -3344.437,E2 -3344.437} C_VEL
LIN {X 0,Y 553.529,Z 531.074,A -85,B 0,C 180,E1 -3344.963,E2 -3344.963} C_VEL
LIN {X 0,Y 553.65,Z 517.426,A -85,B 0,C 180,E1 -3345.367,E2 -3345.367} C_VEL
LIN {X 0,Y 553.528,Z 508.603,A -85,B 0,C 180,E1 -3345.559,E2 -3345.559} C_VEL
LIN {X 0,Y 552.039,Z 501.081,A -85,B 0,C 180,E1 -3345.72,E2 -3345.72} C_VEL
LIN {X 0,Y 552.229,Z 489.47,A -85,B 0,C 180,E1 -3348.553,E2 -3348.553} C_VEL
LIN {X 0,Y 552.379,Z 476.584,A -85,B 0,C 180,E1 -3351.753,E2 -3351.753} C_VEL
LIN {X 0,Y 552.54,Z 465.874,A -85,B 0,C 180,E1 -3354.418,E2 -3354.418} C_VEL
LIN {X 0,Y 552.74,Z 455.404,A -85,B 0,C 180,E1 -3357.122,E2 -3357.122} C_VEL
LIN {X 0,Y 553.091,Z 444.103,A -85,B 0,C 180,E1 -3360.224,E2 -3360.224} C_VEL
LIN {X 0,Y 553.326,Z 437.313,A -85,B 0,C 180,E1 -3362.24,E2 -3362.24} C_VEL
LIN {X 0,Y 552.382,Z 431.622,A -85,B 0,C 180,E1 -3364.208,E2 -3364.208} C_VEL
LIN {X 0,Y 552.134,Z 430.338,A -85,B 0,C 180,E1 -3364.74,E2 -3364.74} C_VEL
LIN {X 0,Y 552.102,Z 430.34,A -85,B 0,C 180,E1 -3367.886,E2 -3367.886} C_VEL
LIN {X 0,Y 552.124,Z 430.339,A -85,B 0,C 180,E1 -3370.481,E2 -3370.481} C_VEL
LIN {X 0,Y 552.111,Z 430.341,A -85,B 0,C 180,E1 -3373.424,E2 -3373.424} C_VEL
LIN {X 0,Y 552.124,Z 430.338,A -85,B 0,C 180,E1 -3376.578,E2 -3376.578} C_VEL
LIN {X 0,Y 552.114,Z 430.34,A -85,B 0,C 180,E1 -3379.519,E2 -3379.519} C_VEL
LIN {X 0,Y 552.097,Z 430.343,A -85,B 0,C 180,E1 -3382.336,E2 -3382.336} C_VEL
LIN {X 0,Y 552.171,Z 430.427,A -85,B 0,C 180,E1 -3384.05,E2 -3384.05} C_VEL
LIN {X 0,Y 552.282,Z 433.849,A -85,B 0,C 180,E1 -3385.808,E2 -3385.808} C_VEL
LIN {X 0,Y 552.158,Z 439.364,A -85,B 0,C 180,E1 -3388.543,E2 -3388.543} C_VEL
LIN {X 0,Y 552.099,Z 445.329,A -85,B 0,C 180,E1 -3391.444,E2 -3391.444} C_VEL
LIN {X 0,Y 552.017,Z 451.5,A -85,B 0,C 180,E1 -3394.35,E2 -3394.35} C_VEL
LIN {X 0,Y 551.933,Z 458.09,A -85,B 0,C 180,E1 -3397.542,E2 -3397.542} C_VEL
LIN {X 0,Y 551.847,Z 464.735,A -85,B 0,C 180,E1 -3400.663,E2 -3400.663} C_VEL
LIN {X 0,Y 551.827,Z 469.884,A -85,B 0,C 180,E1 -3402.967,E2 -3402.967} C_VEL
LIN {X 0,Y 551.763,Z 476.749,A -85,B 0,C 180,E1 -3405.995,E2 -3405.995} C_VEL
LIN {X 0,Y 551.739,Z 479.226,A -85,B 0,C 180,E1 -3407.073,E2 -3407.073} C_VEL
LIN {X 0,Y 553.069,Z 487.912,A -85,B 0,C 180,E1 -3407.291,E2 -3407.291} C_VEL
LIN {X 0,Y 552.893,Z 501.309,A -85,B 0,C 180,E1 -3407.707,E2 -3407.707} C_VEL
LIN {X 0,Y 552.719,Z 513.82,A -85,B 0,C 180,E1 -3408.262,E2 -3408.262} C_VEL
LIN {X 0,Y 552.582,Z 525.259,A -85,B 0,C 180,E1 -3408.927,E2 -3408.927} C_VEL
LIN {X 0,Y 552.37,Z 536.359,A -85,B 0,C 180,E1 -3409.739,E2 -3409.739} C_VEL
LIN {X 0,Y 552.175,Z 546.401,A -85,B 0,C 180,E1 -3410.661,E2 -3410.661} C_VEL
LIN {X 0,Y 552.008,Z 556.1,A -85,B 0,C 180,E1 -3411.765,E2 -3411.765} C_VEL
LIN {X 0,Y 551.896,Z 563.96,A -85,B 0,C 180,E1 -3412.886,E2 -3412.886} C_VEL
LIN {X 0,Y 551.868,Z 570.957,A -85,B 0,C 180,E1 -3414.153,E2 -3414.153} C_VEL
LIN {X 0,Y 551.725,Z 575.697,A -85,B 0,C 180,E1 -3415.251,E2 -3415.251} C_VEL
LIN {X 0,Y 551.751,Z 579.33,A -85,B 0,C 180,E1 -3416.349,E2 -3416.349} C_VEL
LIN {X 0,Y 551.724,Z 581.206,A -85,B 0,C 180,E1 -3417.079,E2 -3417.079} C_VEL
LIN {X 0,Y 551.656,Z 582.629,A -85,B 0,C 180,E1 -3417.81,E2 -3417.81} C_VEL
LIN {X 0,Y 551.642,Z 584.257,A -85,B 0,C 180,E1 -3419.27,E2 -3419.27} C_VEL
LIN {X 0,Y 551.641,Z 584.496,A -85,B 0,C 180,E1 -3420,E2 -3420} C_VEL
LIN {X 0,Y 551.642,Z 584.314,A -85,B 0,C 180,E1 -3420.73,E2 -3420.73} C_VEL
LIN {X 0,Y 551.655,Z 582.765,A -85,B 0,C 180,E1 -3422.19,E2 -3422.19} C_VEL
LIN {X 0,Y 551.724,Z 581.404,A -85,B 0,C 180,E1 -3422.921,E2 -3422.921} C_VEL
LIN {X 0,Y 551.764,Z 578.526,A -85,B 0,C 180,E1 -3424.017,E2 -3424.017} C_VEL
LIN {X 0,Y 551.724,Z 574.624,A -85,B 0,C 180,E1 -3425.116,E2 -3425.116} C_VEL
LIN {X 0,Y 551.811,Z 568.899,A -85,B 0,C 180,E1 -3426.348,E2 -3426.348} C_VEL
LIN {X 0,Y 551.926,Z 562.037,A -85,B 0,C 180,E1 -3427.5,E2 -3427.5} C_VEL
LIN {X 0,Y 552.063,Z 553.854,A -85,B 0,C 180,E1 -3428.603,E2 -3428.603} C_VEL
LIN {X 0,Y 552.197,Z 545.486,A -85,B 0,C 180,E1 -3429.524,E2 -3429.524} C_VEL
LIN {X 0,Y 552.402,Z 535.164,A -85,B 0,C 180,E1 -3430.445,E2 -3430.445} C_VEL
LIN {X 0,Y 552.587,Z 523.322,A -85,B 0,C 180,E1 -3431.289,E2 -3431.289} C_VEL
LIN {X 0,Y 552.752,Z 511.941,A -85,B 0,C 180,E1 -3431.924,E2 -3431.924} C_VEL
LIN {X 0,Y 552.907,Z 499.928,A -85,B 0,C 180,E1 -3432.433,E2 -3432.433} C_VEL
LIN {X 0,Y 552.98,Z 486.524,A -85,B 0,C 180,E1 -3432.836,E2 -3432.836} C_VEL
LIN {X 0,Y 551.747,Z 479.207,A -85,B 0,C 180,E1 -3433.021,E2 -3433.021} C_VEL
LIN {X 0,Y 551.781,Z 473.52,A -85,B 0,C 180,E1 -3435.514,E2 -3435.514} C_VEL
LIN {X 0,Y 551.83,Z 468.369,A -85,B 0,C 180,E1 -3437.798,E2 -3437.798} C_VEL
LIN {X 0,Y 551.843,Z 463.226,A -85,B 0,C 180,E1 -3440.112,E2 -3440.112} C_VEL
LIN {X 0,Y 551.908,Z 458.162,A -85,B 0,C 180,E1 -3442.459,E2 -3442.459} C_VEL
LIN {X 0,Y 551.982,Z 452.063,A -85,B 0,C 180,E1 -3445.311,E2 -3445.311} C_VEL
LIN {X 0,Y 552.048,Z 445.718,A -85,B 0,C 180,E1 -3448.329,E2 -3448.329} C_VEL
LIN {X 0,Y 551.426,Z 444.553,A -85,B 0,C 180,E1 -3448.926,E2 -3448.926} C_VEL
LIN {X 0,Y 548.576,Z 442.905,A -85,B 0,C 180,E1 -3449.901,E2 -3449.901} C_VEL
LIN {X 0,Y 546.161,Z 441.62,A -85,B 0,C 180,E1 -3450.686,E2 -3450.686} C_VEL
LIN {X 0,Y 545.152,Z 440.522,A -85,B 0,C 180,E1 -3451.289,E2 -3451.289} C_VEL
LIN {X 0,Y 545.086,Z 440.118,A -85,B 0,C 180,E1 -3451.493,E2 -3451.493} C_VEL
LIN {X 0,Y 545.168,Z 434.288,A -85,B 0,C 180,E1 -3454.405,E2 -3454.405} C_VEL
LIN {X 0,Y 545.119,Z 431.212,A -85,B 0,C 180,E1 -3456.001,E2 -3456.001} C_VEL
LIN {X 0,Y 545.106,Z 431.212,A -85,B 0,C 180,E1 -3459.323,E2 -3459.323} C_VEL
LIN {X 0,Y 545.087,Z 431.213,A -85,B 0,C 180,E1 -3462.102,E2 -3462.102} C_VEL
LIN {X 0,Y 545.068,Z 431.218,A -85,B 0,C 180,E1 -3465.167,E2 -3465.167} C_VEL
LIN {X 0,Y 545.082,Z 431.216,A -85,B 0,C 180,E1 -3467.897,E2 -3467.897} C_VEL
LIN {X 0,Y 545.092,Z 431.214,A -85,B 0,C 180,E1 -3470.818,E2 -3470.818} C_VEL
LIN {X 0,Y 545.146,Z 431.315,A -85,B 0,C 180,E1 -3471.711,E2 -3471.711} C_VEL
LIN {X 0,Y 545.282,Z 436.787,A -85,B 0,C 180,E1 -3473.637,E2 -3473.637} C_VEL
LIN {X 0,Y 545.229,Z 445.793,A -85,B 0,C 180,E1 -3476.914,E2 -3476.914} C_VEL
LIN {X 0,Y 545.167,Z 454.816,A -85,B 0,C 180,E1 -3480.242,E2 -3480.242} C_VEL
LIN {X 0,Y 545.145,Z 462.906,A -85,B 0,C 180,E1 -3483.177,E2 -3483.177} C_VEL
LIN {X 0,Y 545.072,Z 471.469,A -85,B 0,C 180,E1 -3486.271,E2 -3486.271} C_VEL
LIN {X 0,Y 544.986,Z 478.584,A -85,B 0,C 180,E1 -3488.833,E2 -3488.833} C_VEL
LIN {X 0,Y 544.897,Z 485.019,A -85,B 0,C 180,E1 -3491.188,E2 -3491.188} C_VEL
LIN {X 0,Y 544.844,Z 493.316,A -85,B 0,C 180,E1 -3494.147,E2 -3494.147} C_VEL
LIN {X 0,Y 546.848,Z 504.233,A -85,B 0,C 180,E1 -3494.405,E2 -3494.405} C_VEL
LIN {X 0,Y 546.686,Z 517.833,A -85,B 0,C 180,E1 -3494.782,E2 -3494.782} C_VEL
LIN {X 0,Y 546.446,Z 529.875,A -85,B 0,C 180,E1 -3495.237,E2 -3495.237} C_VEL
LIN {X 0,Y 546.274,Z 540.709,A -85,B 0,C 180,E1 -3495.755,E2 -3495.755} C_VEL
LIN {X 0,Y 545.934,Z 553.45,A -85,B 0,C 180,E1 -3496.506,E2 -3496.506} C_VEL
LIN {X 0,Y 545.668,Z 566.037,A -85,B 0,C 180,E1 -3497.446,E2 -3497.446} C_VEL
LIN {X 0,Y 545.457,Z 575.542,A -85,B 0,C 180,E1 -3498.303,E2 -3498.303} C_VEL
LIN {X 0,Y 545.265,Z 584.257,A -85,B 0,C 180,E1 -3499.228,E2 -3499.228} C_VEL
LIN {X 0,Y 545.061,Z 591.809,A -85,B 0,C 180,E1 -3500.162,E2 -3500.162} C_VEL
LIN {X 0,Y 544.912,Z 599.476,A -85,B 0,C 180,E1 -3501.283,E2 -3501.283} C_VEL
LIN {X 0,Y 544.785,Z 606.849,A -85,B 0,C 180,E1 -3502.587,E2 -3502.587} C_VEL
LIN {X 0,Y 544.732,Z 613.376,A -85,B 0,C 180,E1 -3504.075,E2 -3504.075} C_VEL
LIN {X 0,Y 544.621,Z 617.206,A -85,B 0,C 180,E1 -3505.188,E2 -3505.188} C_VEL
LIN {X 0,Y 544.658,Z 620.193,A -85,B 0,C 180,E1 -3506.3,E2 -3506.3} C_VEL
LIN {X 0,Y 544.647,Z 621.755,A -85,B 0,C 180,E1 -3507.04,E2 -3507.04} C_VEL
LIN {X 0,Y 544.544,Z 623.775,A -85,B 0,C 180,E1 -3508.52,E2 -3508.52} C_VEL
LIN {X 0,Y 544.54,Z 624.443,A -85,B 0,C 180,E1 -3509.999,E2 -3509.999} C_VEL
LIN {X 0,Y 544.538,Z 624.348,A -85,B 0,C 180,E1 -3510.739,E2 -3510.739} C_VEL
LIN {X 0,Y 544.569,Z 623.023,A -85,B 0,C 180,E1 -3512.218,E2 -3512.218} C_VEL
LIN {X 0,Y 544.645,Z 621.932,A -85,B 0,C 180,E1 -3512.958,E2 -3512.958} C_VEL
LIN {X 0,Y 544.655,Z 618.553,A -85,B 0,C 180,E1 -3514.439,E2 -3514.439} C_VEL
LIN {X 0,Y 544.719,Z 615.09,A -85,B 0,C 180,E1 -3515.552,E2 -3515.552} C_VEL
LIN {X 0,Y 544.754,Z 610.719,A -85,B 0,C 180,E1 -3516.667,E2 -3516.667} C_VEL
LIN {X 0,Y 544.819,Z 605.342,A -85,B 0,C 180,E1 -3517.783,E2 -3517.783} C_VEL
LIN {X 0,Y 544.93,Z 598.869,A -85,B 0,C 180,E1 -3518.902,E2 -3518.902} C_VEL
LIN {X 0,Y 545.039,Z 592.493,A -85,B 0,C 180,E1 -3519.836,E2 -3519.836} C_VEL
LIN {X 0,Y 545.222,Z 585.05,A -85,B 0,C 180,E1 -3520.771,E2 -3520.771} C_VEL
LIN {X 0,Y 545.408,Z 576.702,A -85,B 0,C 180,E1 -3521.672,E2 -3521.672} C_VEL
LIN {X 0,Y 545.663,Z 567.102,A -85,B 0,C 180,E1 -3522.552,E2 -3522.552} C_VEL
LIN {X 0,Y 545.879,Z 556.134,A -85,B 0,C 180,E1 -3523.399,E2 -3523.399} C_VEL
LIN {X 0,Y 546.211,Z 542.456,A -85,B 0,C 180,E1 -3524.244,E2 -3524.244} C_VEL
LIN {X 0,Y 546.414,Z 530.903,A -85,B 0,C 180,E1 -3524.81,E2 -3524.81} C_VEL
LIN {X 0,Y 546.63,Z 518.864,A -85,B 0,C 180,E1 -3525.274,E2 -3525.274} C_VEL
LIN {X 0,Y 546.828,Z 506.528,A -85,B 0,C 180,E1 -3525.627,E2 -3525.627} C_VEL
LIN {X 0,Y 546.717,Z 502.509,A -85,B 0,C 180,E1 -3525.726,E2 -3525.726} C_VEL
LIN {X 0,Y 544.814,Z 493.158,A -85,B 0,C 180,E1 -3525.957,E2 -3525.957} C_VEL
LIN {X 0,Y 544.893,Z 485.271,A -85,B 0,C 180,E1 -3528.81,E2 -3528.81} C_VEL
LIN {X 0,Y 544.981,Z 478.837,A -85,B 0,C 180,E1 -3531.166,E2 -3531.166} C_VEL
LIN {X 0,Y 545.071,Z 471.732,A -85,B 0,C 180,E1 -3533.729,E2 -3533.729} C_VEL
LIN {X 0,Y 545.14,Z 463.195,A -85,B 0,C 180,E1 -3536.821,E2 -3536.821} C_VEL
LIN {X 0,Y 545.2,Z 455.082,A -85,B 0,C 180,E1 -3539.754,E2 -3539.754} C_VEL
LIN {X 0,Y 545.234,Z 446.04,A -85,B 0,C 180,E1 -3543.087,E2 -3543.087} C_VEL
LIN {X 0,Y 545.26,Z 438.876,A -85,B 0,C 180,E1 -3545.706,E2 -3545.706} C_VEL
LIN {X 0,Y 545.229,Z 431.945,A -85,B 0,C 180,E1 -3548.16,E2 -3548.16} C_VEL
LIN {X 0,Y 545.133,Z 431.209,A -85,B 0,C 180,E1 -3548.465,E2 -3548.465} C_VEL
LIN {X 0,Y 545.089,Z 431.21,A -85,B 0,C 180,E1 -3551.599,E2 -3551.599} C_VEL
LIN {X 0,Y 545.053,Z 431.218,A -85,B 0,C 180,E1 -3554.128,E2 -3554.128} C_VEL
LIN {X 0,Y 545.083,Z 431.21,A -85,B 0,C 180,E1 -3556.894,E2 -3556.894} C_VEL
LIN {X 0,Y 545.085,Z 431.212,A -85,B 0,C 180,E1 -3559.859,E2 -3559.859} C_VEL
LIN {X 0,Y 545.068,Z 431.217,A -85,B 0,C 180,E1 -3563.072,E2 -3563.072} C_VEL
LIN {X 0,Y 545.082,Z 431.208,A -85,B 0,C 180,E1 -3565.604,E2 -3565.604} C_VEL
LIN {X 0,Y 545.07,Z 431.215,A -85,B 0,C 180,E1 -3568.317,E2 -3568.317} C_VEL
LIN {X 0,Y 545.084,Z 431.211,A -85,B 0,C 180,E1 -3571.25,E2 -3571.25} C_VEL
LIN {X 0,Y 545.08,Z 431.21,A -85,B 0,C 180,E1 -3573.999,E2 -3573.999} C_VEL
LIN {X 0,Y 545.105,Z 431.208,A -85,B 0,C 180,E1 -3576.442,E2 -3576.442} C_VEL
LIN {X 0,Y 545.09,Z 431.208,A -85,B 0,C 180,E1 -3579.628,E2 -3579.628} C_VEL
LIN {X 0,Y 545.087,Z 431.209,A -85,B 0,C 180,E1 -3582.75,E2 -3582.75} C_VEL
LIN {X 0,Y 545.086,Z 431.213,A -85,B 0,C 180,E1 -3585.82,E2 -3585.82} C_VEL
LIN {X 0,Y 545.134,Z 431.206,A -85,B 0,C 180,E1 -3588.85,E2 -3588.85} C_VEL
LIN {X 0,Y 545.127,Z 431.203,A -85,B 0,C 180,E1 -3591.847,E2 -3591.847} C_VEL
LIN {X 0,Y 545.203,Z 431.194,A -85,B 0,C 180,E1 -3594.823,E2 -3594.823} C_VEL
LIN {X 0,Y 545.186,Z 431.201,A -85,B 0,C 180,E1 -3597.784,E2 -3597.784} C_VEL
LIN {X 0,Y 545.207,Z 431.196,A -85,B 0,C 180,E1 -3600.739,E2 -3600.739} C_VEL
LIN {X 0,Y 545.17,Z 431.199,A -85,B 0,C 180,E1 -3602.956,E2 -3602.956} C_VEL
LIN {X 0,Y 545.165,Z 431.199,A -85,B 0,C 180,E1 -3605.92,E2 -3605.92} C_VEL
LIN {X 0,Y 545.12,Z 431.203,A -85,B 0,C 180,E1 -3608.9,E2 -3608.9} C_VEL
LIN {X 0,Y 545.126,Z 431.205,A -85,B 0,C 180,E1 -3611.904,E2 -3611.904} C_VEL
LIN {X 0,Y 545.076,Z 431.216,A -85,B 0,C 180,E1 -3614.944,E2 -3614.944} C_VEL
LIN {X 0,Y 545.074,Z 431.207,A -85,B 0,C 180,E1 -3618.026,E2 -3618.026} C_VEL
LIN {X 0,Y 545.09,Z 431.214,A -85,B 0,C 180,E1 -3620.372,E2 -3620.372} C_VEL
LIN {X 0,Y 545.083,Z 431.214,A -85,B 0,C 180,E1 -3623.559,E2 -3623.559} C_VEL
LIN {X 0,Y 545.08,Z 431.21,A -85,B 0,C 180,E1 -3626.001,E2 -3626.001} C_VEL
LIN {X 0,Y 545.084,Z 431.214,A -85,B 0,C 180,E1 -3628.75,E2 -3628.75} C_VEL
LIN {X 0,Y 545.069,Z 431.211,A -85,B 0,C 180,E1 -3631.683,E2 -3631.683} C_VEL
LIN {X 0,Y 545.076,Z 431.212,A -85,B 0,C 180,E1 -3634.563,E2 -3634.563} C_VEL
LIN {X 0,Y 545.032,Z 431.219,A -85,B 0,C 180,E1 -3637.304,E2 -3637.304} C_VEL
LIN {X 0,Y 545.086,Z 431.209,A -85,B 0,C 180,E1 -3640.141,E2 -3640.141} C_VEL
LIN {X 0,Y 545.062,Z 431.219,A -85,B 0,C 180,E1 -3642.699,E2 -3642.699} C_VEL
LIN {X 0,Y 545.055,Z 431.213,A -85,B 0,C 180,E1 -3645.168,E2 -3645.168} C_VEL
LIN {X 0,Y 545.077,Z 431.217,A -85,B 0,C 180,E1 -3647.899,E2 -3647.899} C_VEL
LIN {X 0,Y 545.101,Z 431.208,A -85,B 0,C 180,E1 -3650.677,E2 -3650.677} C_VEL
LIN {X 0,Y 545.051,Z 431.217,A -85,B 0,C 180,E1 -3653.622,E2 -3653.622} C_VEL
LIN {X 0,Y 545.121,Z 431.378,A -85,B 0,C 180,E1 -3655.672,E2 -3655.672} C_VEL
LIN {X 0,Y 546.255,Z 438.168,A -85,B 0,C 180,E1 -3657.731,E2 -3657.731} C_VEL
LIN {X 0,Y 546.014,Z 447.377,A -85,B 0,C 180,E1 -3660.295,E2 -3660.295} C_VEL
LIN {X 0,Y 545.761,Z 458.211,A -85,B 0,C 180,E1 -3663.212,E2 -3663.212} C_VEL
LIN {X 0,Y 545.519,Z 469.437,A -85,B 0,C 180,E1 -3666.164,E2 -3666.164} C_VEL
LIN {X 0,Y 545.28,Z 481.673,A -85,B 0,C 180,E1 -3669.242,E2 -3669.242} C_VEL
LIN {X 0,Y 545.151,Z 492.6,A -85,B 0,C 180,E1 -3671.978,E2 -3671.978} C_VEL
LIN {X 0,Y 545.019,Z 501.089,A -85,B 0,C 180,E1 -3674.074,E2 -3674.074} C_VEL
LIN {X 0,Y 546.904,Z 511.076,A -85,B 0,C 180,E1 -3674.297,E2 -3674.297} C_VEL
LIN {X 0,Y 546.682,Z 525.886,A -85,B 0,C 180,E1 -3674.671,E2 -3674.671} C_VEL
LIN {X 0,Y 546.438,Z 539.991,A -85,B 0,C 180,E1 -3675.191,E2 -3675.191} C_VEL
LIN {X 0,Y 546.231,Z 553.417,A -85,B 0,C 180,E1 -3675.851,E2 -3675.851} C_VEL
LIN {X 0,Y 545.917,Z 565.532,A -85,B 0,C 180,E1 -3676.602,E2 -3676.602} C_VEL
LIN {X 0,Y 545.625,Z 577.761,A -85,B 0,C 180,E1 -3677.542,E2 -3677.542} C_VEL
LIN {X 0,Y 545.404,Z 588.096,A -85,B 0,C 180,E1 -3678.507,E2 -3678.507} C_VEL
LIN {X 0,Y 545.174,Z 597.861,A -85,B 0,C 180,E1 -3679.603,E2 -3679.603} C_VEL
LIN {X 0,Y 544.999,Z 606.181,A -85,B 0,C 180,E1 -3680.725,E2 -3680.725} C_VEL
LIN {X 0,Y 544.833,Z 614.133,A -85,B 0,C 180,E1 -3682.03,E2 -3682.03} C_VEL
LIN {X 0,Y 544.752,Z 620.88,A -85,B 0,C 180,E1 -3683.414,E2 -3683.414} C_VEL
LIN {X 0,Y 544.645,Z 626.204,A -85,B 0,C 180,E1 -3684.819,E2 -3684.819} C_VEL
LIN {X 0,Y 544.657,Z 630.318,A -85,B 0,C 180,E1 -3686.302,E2 -3686.302} C_VEL
LIN {X 0,Y 544.569,Z 633.003,A -85,B 0,C 180,E1 -3687.782,E2 -3687.782} C_VEL
LIN {X 0,Y 544.539,Z 634.334,A -85,B 0,C 180,E1 -3689.261,E2 -3689.261} C_VEL
LIN {X 0,Y 544.539,Z 634.333,A -85,B 0,C 180,E1 -3690.74,E2 -3690.74} C_VEL
LIN {X 0,Y 544.569,Z 633.002,A -85,B 0,C 180,E1 -3692.22,E2 -3692.22} C_VEL
LIN {X 0,Y 544.657,Z 630.317,A -85,B 0,C 180,E1 -3693.7,E2 -3693.7} C_VEL
LIN {X 0,Y 544.646,Z 626.199,A -85,B 0,C 180,E1 -3695.183,E2 -3695.183} C_VEL
LIN {X 0,Y 544.734,Z 620.949,A -85,B 0,C 180,E1 -3696.57,E2 -3696.57} C_VEL
LIN {X 0,Y 544.834,Z 614.123,A -85,B 0,C 180,E1 -3697.972,E2 -3697.972} C_VEL
LIN {X 0,Y 544.999,Z 606.168,A -85,B 0,C 180,E1 -3699.277,E2 -3699.277} C_VEL
LIN {X 0,Y 545.176,Z 597.845,A -85,B 0,C 180,E1 -3700.398,E2 -3700.398} C_VEL
LIN {X 0,Y 545.366,Z 588.022,A -85,B 0,C 180,E1 -3701.502,E2 -3701.502} C_VEL
LIN {X 0,Y 545.669,Z 576.634,A -85,B 0,C 180,E1 -3702.554,E2 -3702.554} C_VEL
LIN {X 0,Y 545.914,Z 564.091,A -85,B 0,C 180,E1 -3703.494,E2 -3703.494} C_VEL
LIN {X 0,Y 546.283,Z 551.626,A -85,B 0,C 180,E1 -3704.244,E2 -3704.244} C_VEL
LIN {X 0,Y 546.483,Z 538.808,A -85,B 0,C 180,E1 -3704.858,E2 -3704.858} C_VEL
LIN {X 0,Y 546.699,Z 524.532,A -85,B 0,C 180,E1 -3705.37,E2 -3705.37} C_VEL
LIN {X 0,Y 546.837,Z 510.457,A -85,B 0,C 180,E1 -3705.718,E2 -3705.718} C_VEL
LIN {X 0,Y 545.015,Z 501.081,A -85,B 0,C 180,E1 -3705.928,E2 -3705.928} C_VEL
LIN {X 0,Y 545.174,Z 491.031,A -85,B 0,C 180,E1 -3708.412,E2 -3708.412} C_VEL
LIN {X 0,Y 545.36,Z 478.582,A -85,B 0,C 180,E1 -3711.525,E2 -3711.525} C_VEL
LIN {X 0,Y 545.507,Z 467.252,A -85,B 0,C 180,E1 -3714.348,E2 -3714.348} C_VEL
LIN {X 0,Y 545.735,Z 457.991,A -85,B 0,C 180,E1 -3716.791,E2 -3716.791} C_VEL
LIN {X 0,Y 546.136,Z 445.996,A -85,B 0,C 180,E1 -3720.125,E2 -3720.125} C_VEL
LIN {X 0,Y 546.413,Z 438.98,A -85,B 0,C 180,E1 -3722.261,E2 -3722.261} C_VEL
LIN {X 0,Y 545.641,Z 433.945,A -85,B 0,C 180,E1 -3724.03,E2 -3724.03} C_VEL
LIN {X 0,Y 545.084,Z 431.215,A -85,B 0,C 180,E1 -3725.126,E2 -3725.126} C_VEL
LIN {X 0,Y 545.056,Z 431.217,A -85,B 0,C 180,E1 -3728.137,E2 -3728.137} C_VEL
LIN {X 0,Y 545.094,Z 431.215,A -85,B 0,C 180,E1 -3730.474,E2 -3730.474} C_VEL
LIN {X 0,Y 545.083,Z 431.215,A -85,B 0,C 180,E1 -3733.107,E2 -3733.107} C_VEL
LIN {X 0,Y 545.069,Z 431.218,A -85,B 0,C 180,E1 -3736.225,E2 -3736.225} C_VEL
LIN {X 0,Y 545.091,Z 431.214,A -85,B 0,C 180,E1 -3738.886,E2 -3738.886} C_VEL
LIN {X 0,Y 545.055,Z 431.219,A -85,B 0,C 180,E1 -3741.763,E2 -3741.763} C_VEL
LIN {X 0,Y 545.1,Z 431.295,A -85,B 0,C 180,E1 -3743.809,E2 -3743.809} C_VEL
LIN {X 0,Y 545.338,Z 432.638,A -85,B 0,C 180,E1 -3744.554,E2 -3744.554} C_VEL
LIN {X 0,Y 545.207,Z 437.807,A -85,B 0,C 180,E1 -3747.221,E2 -3747.221} C_VEL
LIN {X 0,Y 545.108,Z 442.992,A -85,B 0,C 180,E1 -3749.813,E2 -3749.813} C_VEL
LIN {X 0,Y 545.033,Z 448.13,A -85,B 0,C 180,E1 -3752.341,E2 -3752.341} C_VEL
LIN {X 0,Y 544.977,Z 453.273,A -85,B 0,C 180,E1 -3754.813,E2 -3754.813} C_VEL
LIN {X 0,Y 544.887,Z 459.918,A -85,B 0,C 180,E1 -3758.035,E2 -3758.035} C_VEL
LIN {X 0,Y 544.8,Z 464.881,A -85,B 0,C 180,E1 -3760.403,E2 -3760.403} C_VEL
LIN {X 0,Y 544.7,Z 471.601,A -85,B 0,C 180,E1 -3763.51,E2 -3763.51} C_VEL
LIN {X 0,Y 544.692,Z 476.75,A -85,B 0,C 180,E1 -3765.809,E2 -3765.809} C_VEL
LIN {X 0,Y 544.662,Z 479.264,A -85,B 0,C 180,E1 -3766.902,E2 -3766.902} C_VEL
LIN {X 0,Y 546.137,Z 488.848,A -85,B 0,C 180,E1 -3767.151,E2 -3767.151} C_VEL
LIN {X 0,Y 545.954,Z 501.325,A -85,B 0,C 180,E1 -3767.548,E2 -3767.548} C_VEL
LIN {X 0,Y 545.764,Z 513.83,A -85,B 0,C 180,E1 -3768.11,E2 -3768.11} C_VEL
LIN {X 0,Y 545.612,Z 525.358,A -85,B 0,C 180,E1 -3768.79,E2 -3768.79} C_VEL
LIN {X 0,Y 545.376,Z 536.367,A -85,B 0,C 180,E1 -3769.606,E2 -3769.606} C_VEL
LIN {X 0,Y 545.158,Z 546.406,A -85,B 0,C 180,E1 -3770.539,E2 -3770.539} C_VEL
LIN {X 0,Y 544.976,Z 556.105,A -85,B 0,C 180,E1 -3771.658,E2 -3771.658} C_VEL
LIN {X 0,Y 544.83,Z 563.852,A -85,B 0,C 180,E1 -3772.775,E2 -3772.775} C_VEL
LIN {X 0,Y 544.778,Z 570.96,A -85,B 0,C 180,E1 -3774.076,E2 -3774.076} C_VEL
LIN {X 0,Y 544.629,Z 575.7,A -85,B 0,C 180,E1 -3775.189,E2 -3775.189} C_VEL
LIN {X 0,Y 544.67,Z 579.332,A -85,B 0,C 180,E1 -3776.301,E2 -3776.301} C_VEL
LIN {X 0,Y 544.651,Z 581.207,A -85,B 0,C 180,E1 -3777.041,E2 -3777.041} C_VEL
LIN {X 0,Y 544.571,Z 582.629,A -85,B 0,C 180,E1 -3777.781,E2 -3777.781} C_VEL
LIN {X 0,Y 544.542,Z 584.258,A -85,B 0,C 180,E1 -3779.261,E2 -3779.261} C_VEL
LIN {X 0,Y 544.541,Z 584.496,A -85,B 0,C 180,E1 -3780,E2 -3780} C_VEL
LIN {X 0,Y 544.542,Z 584.314,A -85,B 0,C 180,E1 -3780.74,E2 -3780.74} C_VEL
LIN {X 0,Y 544.57,Z 582.764,A -85,B 0,C 180,E1 -3782.219,E2 -3782.219} C_VEL
LIN {X 0,Y 544.651,Z 581.402,A -85,B 0,C 180,E1 -3782.959,E2 -3782.959} C_VEL
LIN {X 0,Y 544.684,Z 578.524,A -85,B 0,C 180,E1 -3784.07,E2 -3784.07} C_VEL
LIN {X 0,Y 544.653,Z 574.622,A -85,B 0,C 180,E1 -3785.182,E2 -3785.182} C_VEL
LIN {X 0,Y 544.724,Z 569.403,A -85,B 0,C 180,E1 -3786.334,E2 -3786.334} C_VEL
LIN {X 0,Y 544.86,Z 562.033,A -85,B 0,C 180,E1 -3787.598,E2 -3787.598} C_VEL
LIN {X 0,Y 544.999,Z 553.849,A -85,B 0,C 180,E1 -3788.715,E2 -3788.715} C_VEL
LIN {X 0,Y 545.16,Z 545.48,A -85,B 0,C 180,E1 -3789.648,E2 -3789.648} C_VEL
LIN {X 0,Y 545.379,Z 535.155,A -85,B 0,C 180,E1 -3790.581,E2 -3790.581} C_VEL
LIN {X 0,Y 545.613,Z 523.703,A -85,B 0,C 180,E1 -3791.409,E2 -3791.409} C_VEL
LIN {X 0,Y 545.791,Z 511.93,A -85,B 0,C 180,E1 -3792.078,E2 -3792.078} C_VEL
LIN {X 0,Y 545.994,Z 499.911,A -85,B 0,C 180,E1 -3792.593,E2 -3792.593} C_VEL
LIN {X 0,Y 546.017,Z 487.301,A -85,B 0,C 180,E1 -3792.982,E2 -3792.982} C_VEL
LIN {X 0,Y 544.649,Z 479.206,A -85,B 0,C 180,E1 -3793.193,E2 -3793.193} C_VEL
LIN {X 0,Y 544.687,Z 473.518,A -85,B 0,C 180,E1 -3795.721,E2 -3795.721} C_VEL
LIN {X 0,Y 544.737,Z 468.379,A -85,B 0,C 180,E1 -3798.038,E2 -3798.038} C_VEL
LIN {X 0,Y 544.788,Z 463.306,A -85,B 0,C 180,E1 -3800.384,E2 -3800.384} C_VEL
LIN {X 0,Y 544.853,Z 458.238,A -85,B 0,C 180,E1 -3802.766,E2 -3802.766} C_VEL
LIN {X 0,Y 544.918,Z 452.525,A -85,B 0,C 180,E1 -3805.468,E2 -3805.468} C_VEL
LIN {X 0,Y 545.018,Z 446.232,A -85,B 0,C 180,E1 -3808.497,E2 -3808.497} C_VEL
LIN {X 0,Y 545.086,Z 440.118,A -85,B 0,C 180,E1 -3811.493,E2 -3811.493} C_VEL
LIN {X 0,Y 544.469,Z 438.981,A -85,B 0,C 180,E1 -3812.098,E2 -3812.098} C_VEL
LIN {X 0,Y 541.653,Z 437.394,A -85,B 0,C 180,E1 -3813.086,E2 -3813.086} C_VEL
LIN {X 0,Y 539.247,Z 436.158,A -85,B 0,C 180,E1 -3813.882,E2 -3813.882} C_VEL
LIN {X 0,Y 538.213,Z 435.107,A -85,B 0,C 180,E1 -3814.494,E2 -3814.494} C_VEL
LIN {X 0,Y 538.13,Z 434.718,A -85,B 0,C 180,E1 -3814.701,E2 -3814.701} C_VEL
LIN {X 0,Y 538.065,Z 432.09,A -85,B 0,C 180,E1 -3816.115,E2 -3816.115} C_VEL
LIN {X 0,Y 538.038,Z 432.093,A -85,B 0,C 180,E1 -3819.585,E2 -3819.585} C_VEL
LIN {X 0,Y 538.04,Z 432.092,A -85,B 0,C 180,E1 -3821.879,E2 -3821.879} C_VEL
LIN {X 0,Y 538.038,Z 432.094,A -85,B 0,C 180,E1 -3825.14,E2 -3825.14} C_VEL
LIN {X 0,Y 538.035,Z 432.095,A -85,B 0,C 180,E1 -3828.226,E2 -3828.226} C_VEL
LIN {X 0,Y 538.095,Z 432.096,A -85,B 0,C 180,E1 -3831.596,E2 -3831.596} C_VEL
LIN {X 0,Y 538.267,Z 437.588,A -85,B 0,C 180,E1 -3833.552,E2 -3833.552} C_VEL
LIN {X 0,Y 538.181,Z 446.275,A -85,B 0,C 180,E1 -3836.737,E2 -3836.737} C_VEL
LIN {X 0,Y 538.132,Z 453.786,A -85,B 0,C 180,E1 -3839.538,E2 -3839.538} C_VEL
LIN {X 0,Y 538.088,Z 462.226,A -85,B 0,C 180,E1 -3842.642,E2 -3842.642} C_VEL
LIN {X 0,Y 538.019,Z 470.641,A -85,B 0,C 180,E1 -3845.702,E2 -3845.702} C_VEL
LIN {X 0,Y 537.935,Z 478.463,A -85,B 0,C 180,E1 -3848.542,E2 -3848.542} C_VEL
LIN {X 0,Y 537.84,Z 486.082,A -85,B 0,C 180,E1 -3851.328,E2 -3851.328} C_VEL
LIN {X 0,Y 537.752,Z 493.171,A -85,B 0,C 180,E1 -3853.924,E2 -3853.924} C_VEL
LIN {X 0,Y 539.984,Z 505.001,A -85,B 0,C 180,E1 -3854.222,E2 -3854.222} C_VEL
LIN {X 0,Y 539.836,Z 517.681,A -85,B 0,C 180,E1 -3854.579,E2 -3854.579} C_VEL
LIN {X 0,Y 539.586,Z 528.768,A -85,B 0,C 180,E1 -3854.996,E2 -3854.996} C_VEL
LIN {X 0,Y 539.422,Z 538.899,A -85,B 0,C 180,E1 -3855.474,E2 -3855.474} C_VEL
LIN {X 0,Y 539.115,Z 548.931,A -85,B 0,C 180,E1 -3856.044,E2 -3856.044} C_VEL
LIN {X 0,Y 538.885,Z 558.731,A -85,B 0,C 180,E1 -3856.71,E2 -3856.71} C_VEL
LIN {X 0,Y 538.621,Z 568.223,A -85,B 0,C 180,E1 -3857.471,E2 -3857.471} C_VEL
LIN {X 0,Y 538.409,Z 576.924,A -85,B 0,C 180,E1 -3858.288,E2 -3858.288} C_VEL
LIN {X 0,Y 538.236,Z 585.878,A -85,B 0,C 180,E1 -3859.276,E2 -3859.276} C_VEL
LIN {X 0,Y 537.974,Z 594.582,A -85,B 0,C 180,E1 -3860.411,E2 -3860.411} C_VEL
LIN {X 0,Y 537.816,Z 602.822,A -85,B 0,C 180,E1 -3861.735,E2 -3861.735} C_VEL
LIN {X 0,Y 537.663,Z 608.613,A -85,B 0,C 180,E1 -3862.866,E2 -3862.866} C_VEL
LIN {X 0,Y 537.645,Z 613.372,A -85,B 0,C 180,E1 -3863.996,E2 -3863.996} C_VEL
LIN {X 0,Y 537.533,Z 617.203,A -85,B 0,C 180,E1 -3865.124,E2 -3865.124} C_VEL
LIN {X 0,Y 537.577,Z 620.188,A -85,B 0,C 180,E1 -3866.251,E2 -3866.251} C_VEL
LIN {X 0,Y 537.548,Z 621.758,A -85,B 0,C 180,E1 -3867.001,E2 -3867.001} C_VEL
LIN {X 0,Y 537.45,Z 623.77,A -85,B 0,C 180,E1 -3868.5,E2 -3868.5} C_VEL
LIN {X 0,Y 537.441,Z 624.437,A -85,B 0,C 180,E1 -3869.999,E2 -3869.999} C_VEL
LIN {X 0,Y 537.438,Z 624.346,A -85,B 0,C 180,E1 -3870.748,E2 -3870.748} C_VEL
LIN {X 0,Y 537.488,Z 623.017,A -85,B 0,C 180,E1 -3872.247,E2 -3872.247} C_VEL
LIN {X 0,Y 537.546,Z 621.931,A -85,B 0,C 180,E1 -3872.997,E2 -3872.997} C_VEL
LIN {X 0,Y 537.551,Z 618.547,A -85,B 0,C 180,E1 -3874.498,E2 -3874.498} C_VEL
LIN {X 0,Y 537.649,Z 615.081,A -85,B 0,C 180,E1 -3875.625,E2 -3875.625} C_VEL
LIN {X 0,Y 537.666,Z 610.71,A -85,B 0,C 180,E1 -3876.755,E2 -3876.755} C_VEL
LIN {X 0,Y 537.761,Z 605.334,A -85,B 0,C 180,E1 -3877.886,E2 -3877.886} C_VEL
LIN {X 0,Y 537.867,Z 598.858,A -85,B 0,C 180,E1 -3879.02,E2 -3879.02} C_VEL
LIN {X 0,Y 538.016,Z 592.481,A -85,B 0,C 180,E1 -3879.966,E2 -3879.966} C_VEL
LIN {X 0,Y 538.215,Z 585.039,A -85,B 0,C 180,E1 -3880.913,E2 -3880.913} C_VEL
LIN {X 0,Y 538.396,Z 577.376,A -85,B 0,C 180,E1 -3881.756,E2 -3881.756} C_VEL
LIN {X 0,Y 538.615,Z 569.275,A -85,B 0,C 180,E1 -3882.528,E2 -3882.528} C_VEL
LIN {X 0,Y 538.858,Z 559.957,A -85,B 0,C 180,E1 -3883.288,E2 -3883.288} C_VEL
LIN {X 0,Y 539.074,Z 550.373,A -85,B 0,C 180,E1 -3883.956,E2 -3883.956} C_VEL
LIN {X 0,Y 539.396,Z 540.623,A -85,B 0,C 180,E1 -3884.525,E2 -3884.525} C_VEL
LIN {X 0,Y 539.567,Z 529.768,A -85,B 0,C 180,E1 -3885.051,E2 -3885.051} C_VEL
LIN {X 0,Y 539.776,Z 518.471,A -85,B 0,C 180,E1 -3885.485,E2 -3885.485} C_VEL
LIN {X 0,Y 540.004,Z 505.929,A -85,B 0,C 180,E1 -3885.844,E2 -3885.844} C_VEL
LIN {X 0,Y 539.59,Z 502.045,A -85,B 0,C 180,E1 -3885.948,E2 -3885.948} C_VEL
LIN {X 0,Y 537.745,Z 493.156,A -85,B 0,C 180,E1 -3886.172,E2 -3886.172} C_VEL
LIN {X 0,Y 537.846,Z 485.253,A -85,B 0,C 180,E1 -3889.066,E2 -3889.066} C_VEL
LIN {X 0,Y 537.975,Z 477.358,A -85,B 0,C 180,E1 -3891.947,E2 -3891.947} C_VEL
LIN {X 0,Y 538.024,Z 468.634,A -85,B 0,C 180,E1 -3895.12,E2 -3895.12} C_VEL
LIN {X 0,Y 538.09,Z 462.488,A -85,B 0,C 180,E1 -3897.358,E2 -3897.358} C_VEL
LIN {X 0,Y 538.133,Z 454.041,A -85,B 0,C 180,E1 -3900.463,E2 -3900.463} C_VEL
LIN {X 0,Y 538.201,Z 445.327,A -85,B 0,C 180,E1 -3903.707,E2 -3903.707} C_VEL
LIN {X 0,Y 538.265,Z 437.847,A -85,B 0,C 180,E1 -3906.446,E2 -3906.446} C_VEL
LIN {X 0,Y 538.106,Z 432.084,A -85,B 0,C 180,E1 -3908.522,E2 -3908.522} C_VEL
LIN {X 0,Y 538.072,Z 432.09,A -85,B 0,C 180,E1 -3910.772,E2 -3910.772} C_VEL
LIN {X 0,Y 538.023,Z 432.093,A -85,B 0,C 180,E1 -3914.074,E2 -3914.074} C_VEL
LIN {X 0,Y 538.019,Z 432.091,A -85,B 0,C 180,E1 -3917.214,E2 -3917.214} C_VEL
LIN {X 0,Y 538.047,Z 432.086,A -85,B 0,C 180,E1 -3920.205,E2 -3920.205} C_VEL
LIN {X 0,Y 538.022,Z 432.095,A -85,B 0,C 180,E1 -3923.067,E2 -3923.067} C_VEL
LIN {X 0,Y 538.024,Z 432.087,A -85,B 0,C 180,E1 -3925.827,E2 -3925.827} C_VEL
LIN {X 0,Y 538.016,Z 432.091,A -85,B 0,C 180,E1 -3928.499,E2 -3928.499} C_VEL
LIN {X 0,Y 538.05,Z 432.087,A -85,B 0,C 180,E1 -3931.099,E2 -3931.099} C_VEL
LIN {X 0,Y 538.041,Z 432.09,A -85,B 0,C 180,E1 -3933.633,E2 -3933.633} C_VEL
LIN {X 0,Y 538.032,Z 432.088,A -85,B 0,C 180,E1 -3936.113,E2 -3936.113} C_VEL
LIN {X 0,Y 538.034,Z 432.087,A -85,B 0,C 180,E1 -3939.348,E2 -3939.348} C_VEL
LIN {X 0,Y 538.062,Z 432.086,A -85,B 0,C 180,E1 -3942.517,E2 -3942.517} C_VEL
LIN {X 0,Y 538.054,Z 432.091,A -85,B 0,C 180,E1 -3945.63,E2 -3945.63} C_VEL
LIN {X 0,Y 538.088,Z 432.082,A -85,B 0,C 180,E1 -3948.702,E2 -3948.702} C_VEL
LIN {X 0,Y 538.083,Z 432.08,A -85,B 0,C 180,E1 -3951.739,E2 -3951.739} C_VEL
LIN {X 0,Y 538.179,Z 432.069,A -85,B 0,C 180,E1 -3954.755,E2 -3954.755} C_VEL
LIN {X 0,Y 538.158,Z 432.077,A -85,B 0,C 180,E1 -3957.755,E2 -3957.755} C_VEL
LIN {X 0,Y 538.176,Z 432.072,A -85,B 0,C 180,E1 -3960.748,E2 -3960.748} C_VEL
LIN {X 0,Y 538.136,Z 432.074,A -85,B 0,C 180,E1 -3962.994,E2 -3962.994} C_VEL
LIN {X 0,Y 538.117,Z 432.078,A -85,B 0,C 180,E1 -3965.997,E2 -3965.997} C_VEL
LIN {X 0,Y 538.069,Z 432.081,A -85,B 0,C 180,E1 -3969.018,E2 -3969.018} C_VEL
LIN {X 0,Y 538.074,Z 432.082,A -85,B 0,C 180,E1 -3972.063,E2 -3972.063} C_VEL
LIN {X 0,Y 538.036,Z 432.091,A -85,B 0,C 180,E1 -3975.144,E2 -3975.144} C_VEL
LIN {X 0,Y 538.026,Z 432.087,A -85,B 0,C 180,E1 -3978.27,E2 -3978.27} C_VEL
LIN {X 0,Y 538.033,Z 432.089,A -85,B 0,C 180,E1 -3980.652,E2 -3980.652} C_VEL
LIN {X 0,Y 538.014,Z 432.094,A -85,B 0,C 180,E1 -3983.888,E2 -3983.888} C_VEL
LIN {X 0,Y 538.041,Z 432.086,A -85,B 0,C 180,E1 -3986.367,E2 -3986.367} C_VEL
LIN {X 0,Y 538.047,Z 432.093,A -85,B 0,C 180,E1 -3988.939,E2 -3988.939} C_VEL
LIN {X 0,Y 538.019,Z 432.09,A -85,B 0,C 180,E1 -3991.891,E2 -3991.891} C_VEL
LIN {X 0,Y 538.026,Z 432.09,A -85,B 0,C 180,E1 -3994.622,E2 -3994.622} C_VEL
LIN {X 0,Y 538,Z 432.093,A -85,B 0,C 180,E1 -3997.171,E2 -3997.171} C_VEL
LIN {X 0,Y 538.047,Z 432.087,A -85,B 0,C 180,E1 -3999.795,E2 -3999.795} C_VEL
LIN {X 0,Y 538.019,Z 432.096,A -85,B 0,C 180,E1 -4002.786,E2 -4002.786} C_VEL
LIN {X 0,Y 538.025,Z 432.089,A -85,B 0,C 180,E1 -4005.142,E2 -4005.142} C_VEL
LIN {X 0,Y 538.035,Z 432.092,A -85,B 0,C 180,E1 -4008.229,E2 -4008.229} C_VEL
LIN {X 0,Y 538.054,Z 432.086,A -85,B 0,C 180,E1 -4010.412,E2 -4010.412} C_VEL
LIN {X 0,Y 538.024,Z 432.094,A -85,B 0,C 180,E1 -4013.069,E2 -4013.069} C_VEL
LIN {X 0,Y 538.048,Z 432.169,A -85,B 0,C 180,E1 -4015.377,E2 -4015.377} C_VEL
LIN {X 0,Y 539.174,Z 438.206,A -85,B 0,C 180,E1 -4017.254,E2 -4017.254} C_VEL
LIN {X 0,Y 539.259,Z 442.776,A -85,B 0,C 180,E1 -4018.581,E2 -4018.581} C_VEL
LIN {X 0,Y 538.924,Z 453.517,A -85,B 0,C 180,E1 -4021.578,E2 -4021.578} C_VEL
LIN {X 0,Y 538.647,Z 464.347,A -85,B 0,C 180,E1 -4024.498,E2 -4024.498} C_VEL
LIN {X 0,Y 538.392,Z 475.22,A -85,B 0,C 180,E1 -4027.352,E2 -4027.352} C_VEL
LIN {X 0,Y 538.2,Z 487.887,A -85,B 0,C 180,E1 -4030.551,E2 -4030.551} C_VEL
LIN {X 0,Y 538.019,Z 498.844,A -85,B 0,C 180,E1 -4033.3,E2 -4033.3} C_VEL
LIN {X 0,Y 537.975,Z 501.089,A -85,B 0,C 180,E1 -4033.859,E2 -4033.859} C_VEL
LIN {X 0,Y 540.06,Z 512.218,A -85,B 0,C 180,E1 -4034.117,E2 -4034.117} C_VEL
LIN {X 0,Y 539.822,Z 526.686,A -85,B 0,C 180,E1 -4034.497,E2 -4034.497} C_VEL
LIN {X 0,Y 539.554,Z 541.116,A -85,B 0,C 180,E1 -4035.046,E2 -4035.046} C_VEL
LIN {X 0,Y 539.338,Z 553.419,A -85,B 0,C 180,E1 -4035.666,E2 -4035.666} C_VEL
LIN {X 0,Y 538.959,Z 565.533,A -85,B 0,C 180,E1 -4036.426,E2 -4036.426} C_VEL
LIN {X 0,Y 538.668,Z 577.76,A -85,B 0,C 180,E1 -4037.378,E2 -4037.378} C_VEL
LIN {X 0,Y 538.398,Z 588.702,A -85,B 0,C 180,E1 -4038.42,E2 -4038.42} C_VEL
LIN {X 0,Y 538.153,Z 597.861,A -85,B 0,C 180,E1 -4039.466,E2 -4039.466} C_VEL
LIN {X 0,Y 537.971,Z 606.182,A -85,B 0,C 180,E1 -4040.603,E2 -4040.603} C_VEL
LIN {X 0,Y 537.755,Z 614.133,A -85,B 0,C 180,E1 -4041.925,E2 -4041.925} C_VEL
LIN {X 0,Y 537.685,Z 621.223,A -85,B 0,C 180,E1 -4043.407,E2 -4043.407} C_VEL
LIN {X 0,Y 537.578,Z 626.204,A -85,B 0,C 180,E1 -4044.75,E2 -4044.75} C_VEL
LIN {X 0,Y 537.576,Z 630.318,A -85,B 0,C 180,E1 -4046.253,E2 -4046.253} C_VEL
LIN {X 0,Y 537.488,Z 633.003,A -85,B 0,C 180,E1 -4047.753,E2 -4047.753} C_VEL
LIN {X 0,Y 537.439,Z 634.334,A -85,B 0,C 180,E1 -4049.252,E2 -4049.252} C_VEL
LIN {X 0,Y 537.439,Z 634.333,A -85,B 0,C 180,E1 -4050.75,E2 -4050.75} C_VEL
LIN {X 0,Y 537.488,Z 633.003,A -85,B 0,C 180,E1 -4052.249,E2 -4052.249} C_VEL
LIN {X 0,Y 537.576,Z 630.317,A -85,B 0,C 180,E1 -4053.749,E2 -4053.749} C_VEL
LIN {X 0,Y 537.578,Z 626.199,A -85,B 0,C 180,E1 -4055.252,E2 -4055.252} C_VEL
LIN {X 0,Y 537.667,Z 620.523,A -85,B 0,C 180,E1 -4056.757,E2 -4056.757} C_VEL
LIN {X 0,Y 537.757,Z 614.123,A -85,B 0,C 180,E1 -4058.077,E2 -4058.077} C_VEL
LIN {X 0,Y 537.971,Z 606.169,A -85,B 0,C 180,E1 -4059.399,E2 -4059.399} C_VEL
LIN {X 0,Y 538.155,Z 597.846,A -85,B 0,C 180,E1 -4060.536,E2 -4060.536} C_VEL
LIN {X 0,Y 538.352,Z 588.669,A -85,B 0,C 180,E1 -4061.584,E2 -4061.584} C_VEL
LIN {X 0,Y 538.678,Z 577.737,A -85,B 0,C 180,E1 -4062.624,E2 -4062.624} C_VEL
LIN {X 0,Y 538.962,Z 565.507,A -85,B 0,C 180,E1 -4063.576,E2 -4063.576} C_VEL
LIN {X 0,Y 539.337,Z 553.386,A -85,B 0,C 180,E1 -4064.336,E2 -4064.336} C_VEL
LIN {X 0,Y 539.586,Z 539.936,A -85,B 0,C 180,E1 -4065.004,E2 -4065.004} C_VEL
LIN {X 0,Y 539.835,Z 525.697,A -85,B 0,C 180,E1 -4065.534,E2 -4065.534} C_VEL
LIN {X 0,Y 540.029,Z 511.551,A -85,B 0,C 180,E1 -4065.898,E2 -4065.898} C_VEL
LIN {X 0,Y 537.974,Z 501.081,A -85,B 0,C 180,E1 -4066.143,E2 -4066.143} C_VEL
LIN {X 0,Y 538.167,Z 491.031,A -85,B 0,C 180,E1 -4068.661,E2 -4068.661} C_VEL
LIN {X 0,Y 538.319,Z 478.649,A -85,B 0,C 180,E1 -4071.747,E2 -4071.747} C_VEL
LIN {X 0,Y 538.523,Z 467.084,A -85,B 0,C 180,E1 -4074.685,E2 -4074.685} C_VEL
LIN {X 0,Y 538.828,Z 456.729,A -85,B 0,C 180,E1 -4077.51,E2 -4077.51} C_VEL
LIN {X 0,Y 539.241,Z 445.781,A -85,B 0,C 180,E1 -4080.662,E2 -4080.662} C_VEL
LIN {X 0,Y 539.501,Z 440.639,A -85,B 0,C 180,E1 -4082.284,E2 -4082.284} C_VEL
LIN {X 0,Y 538.738,Z 435.563,A -85,B 0,C 180,E1 -4084.122,E2 -4084.122} C_VEL
LIN {X 0,Y 538.013,Z 432.097,A -85,B 0,C 180,E1 -4085.589,E2 -4085.589} C_VEL
LIN {X 0,Y 538.009,Z 432.095,A -85,B 0,C 180,E1 -4088.392,E2 -4088.392} C_VEL
LIN {X 0,Y 538.055,Z 432.09,A -85,B 0,C 180,E1 -4090.776,E2 -4090.776} C_VEL
LIN {X 0,Y 538.024,Z 432.093,A -85,B 0,C 180,E1 -4094.074,E2 -4094.074} C_VEL
LIN {X 0,Y 538.038,Z 432.091,A -85,B 0,C 180,E1 -4097.012,E2 -4097.012} C_VEL
LIN {X 0,Y 538.053,Z 432.092,A -85,B 0,C 180,E1 -4099.253,E2 -4099.253} C_VEL
LIN {X 0,Y 537.996,Z 432.099,A -85,B 0,C 180,E1 -4102.123,E2 -4102.123} C_VEL
LIN {X 0,Y 538.048,Z 432.166,A -85,B 0,C 180,E1 -4103.536,E2 -4103.536} C_VEL
LIN {X 0,Y 538.311,Z 435.393,A -85,B 0,C 180,E1 -4105.337,E2 -4105.337} C_VEL
LIN {X 0,Y 538.127,Z 440.655,A -85,B 0,C 180,E1 -4108.094,E2 -4108.094} C_VEL
LIN {X 0,Y 538.048,Z 446.587,A -85,B 0,C 180,E1 -4111.099,E2 -4111.099} C_VEL
LIN {X 0,Y 537.933,Z 451.697,A -85,B 0,C 180,E1 -4113.628,E2 -4113.628} C_VEL
LIN {X 0,Y 537.87,Z 456.907,A -85,B 0,C 180,E1 -4116.156,E2 -4116.156} C_VEL
LIN {X 0,Y 537.802,Z 461.748,A -85,B 0,C 180,E1 -4118.537,E2 -4118.537} C_VEL
LIN {X 0,Y 537.701,Z 466.717,A -85,B 0,C 180,E1 -4120.928,E2 -4120.928} C_VEL
LIN {X 0,Y 537.635,Z 471.707,A -85,B 0,C 180,E1 -4123.287,E2 -4123.287} C_VEL
LIN {X 0,Y 537.628,Z 476.751,A -85,B 0,C 180,E1 -4125.619,E2 -4125.619} C_VEL
LIN {X 0,Y 537.581,Z 479.303,A -85,B 0,C 180,E1 -4126.726,E2 -4126.726} C_VEL
LIN {X 0,Y 539.213,Z 489.785,A -85,B 0,C 180,E1 -4127.007,E2 -4127.007} C_VEL
LIN {X 0,Y 539.001,Z 502.54,A -85,B 0,C 180,E1 -4127.433,E2 -4127.433} C_VEL
LIN {X 0,Y 538.815,Z 513.84,A -85,B 0,C 180,E1 -4127.954,E2 -4127.954} C_VEL
LIN {X 0,Y 538.623,Z 524.482,A -85,B 0,C 180,E1 -4128.583,E2 -4128.583} C_VEL
LIN {X 0,Y 538.416,Z 535.211,A -85,B 0,C 180,E1 -4129.375,E2 -4129.375} C_VEL
LIN {X 0,Y 538.166,Z 544.585,A -85,B 0,C 180,E1 -4130.226,E2 -4130.226} C_VEL
LIN {X 0,Y 537.989,Z 553.136,A -85,B 0,C 180,E1 -4131.17,E2 -4131.17} C_VEL
LIN {X 0,Y 537.821,Z 561.443,A -85,B 0,C 180,E1 -4132.303,E2 -4132.303} C_VEL
LIN {X 0,Y 537.687,Z 567.999,A -85,B 0,C 180,E1 -4133.407,E2 -4133.407} C_VEL
LIN {X 0,Y 537.588,Z 574.274,A -85,B 0,C 180,E1 -4134.749,E2 -4134.749} C_VEL
LIN {X 0,Y 537.604,Z 578.262,A -85,B 0,C 180,E1 -4135.877,E2 -4135.877} C_VEL
LIN {X 0,Y 537.552,Z 581.209,A -85,B 0,C 180,E1 -4137.002,E2 -4137.002} C_VEL
LIN {X 0,Y 537.489,Z 582.63,A -85,B 0,C 180,E1 -4137.752,E2 -4137.752} C_VEL
LIN {X 0,Y 537.442,Z 584.258,A -85,B 0,C 180,E1 -4139.251,E2 -4139.251} C_VEL
LIN {X 0,Y 537.442,Z 584.496,A -85,B 0,C 180,E1 -4140,E2 -4140} C_VEL
LIN {X 0,Y 537.442,Z 584.314,A -85,B 0,C 180,E1 -4140.749,E2 -4140.749} C_VEL
LIN {X 0,Y 537.489,Z 582.762,A -85,B 0,C 180,E1 -4142.248,E2 -4142.248} C_VEL
LIN {X 0,Y 537.552,Z 581.4,A -85,B 0,C 180,E1 -4142.998,E2 -4142.998} C_VEL
LIN {X 0,Y 537.604,Z 578.522,A -85,B 0,C 180,E1 -4144.123,E2 -4144.123} C_VEL
LIN {X 0,Y 537.587,Z 574.62,A -85,B 0,C 180,E1 -4145.251,E2 -4145.251} C_VEL
LIN {X 0,Y 537.636,Z 569.876,A -85,B 0,C 180,E1 -4146.319,E2 -4146.319} C_VEL
LIN {X 0,Y 537.791,Z 563.256,A -85,B 0,C 180,E1 -4147.509,E2 -4147.509} C_VEL
LIN {X 0,Y 537.953,Z 555.33,A -85,B 0,C 180,E1 -4148.641,E2 -4148.641} C_VEL
LIN {X 0,Y 538.133,Z 545.474,A -85,B 0,C 180,E1 -4149.775,E2 -4149.775} C_VEL
LIN {X 0,Y 538.376,Z 535.146,A -85,B 0,C 180,E1 -4150.721,E2 -4150.721} C_VEL
LIN {X 0,Y 538.64,Z 524.015,A -85,B 0,C 180,E1 -4151.538,E2 -4151.538} C_VEL
LIN {X 0,Y 538.82,Z 513.736,A -85,B 0,C 180,E1 -4152.141,E2 -4152.141} C_VEL
LIN {X 0,Y 539.03,Z 501.194,A -85,B 0,C 180,E1 -4152.71,E2 -4152.71} C_VEL
LIN {X 0,Y 539.098,Z 488.193,A -85,B 0,C 180,E1 -4153.128,E2 -4153.128} C_VEL
LIN {X 0,Y 537.592,Z 479.204,A -85,B 0,C 180,E1 -4153.37,E2 -4153.37} C_VEL
LIN {X 0,Y 537.619,Z 473.539,A -85,B 0,C 180,E1 -4155.934,E2 -4155.934} C_VEL
LIN {X 0,Y 537.66,Z 468.457,A -85,B 0,C 180,E1 -4158.283,E2 -4158.283} C_VEL
LIN {X 0,Y 537.736,Z 463.403,A -85,B 0,C 180,E1 -4160.664,E2 -4160.664} C_VEL
LIN {X 0,Y 537.779,Z 458.309,A -85,B 0,C 180,E1 -4163.083,E2 -4163.083} C_VEL
LIN {X 0,Y 537.866,Z 452.982,A -85,B 0,C 180,E1 -4165.632,E2 -4165.632} C_VEL
LIN {X 0,Y 537.996,Z 446.219,A -85,B 0,C 180,E1 -4168.926,E2 -4168.926} C_VEL
LIN {X 0,Y 538.064,Z 440.237,A -85,B 0,C 180,E1 -4171.895,E2 -4171.895} C_VEL
LIN {X 0,Y 538.13,Z 434.718,A -85,B 0,C 180,E1 -4174.701,E2 -4174.701} C_VEL
LIN {X 0,Y 537.45,Z 433.767,A -85,B 0,C 180,E1 -4175.316,E2 -4175.316} C_VEL
LIN {X 0,Y 534.543,Z 433.047,A -85,B 0,C 180,E1 -4176.326,E2 -4176.326} C_VEL
LIN {X 0,Y 532.085,Z 432.947,A -85,B 0,C 180,E1 -4177.144,E2 -4177.144} C_VEL
LIN {X 0,Y 531.032,Z 432.97,A -85,B 0,C 180,E1 -4177.776,E2 -4177.776} C_VEL
LIN {X 0,Y 530.947,Z 432.974,A -85,B 0,C 180,E1 -4177.99,E2 -4177.99} C_VEL
LIN {X 0,Y 530.987,Z 432.97,A -85,B 0,C 180,E1 -4180.433,E2 -4180.433} C_VEL
LIN {X 0,Y 530.976,Z 432.971,A -85,B 0,C 180,E1 -4183.282,E2 -4183.282} C_VEL
LIN {X 0,Y 530.99,Z 432.97,A -85,B 0,C 180,E1 -4185.621,E2 -4185.621} C_VEL
LIN {X 0,Y 530.998,Z 432.97,A -85,B 0,C 180,E1 -4188.564,E2 -4188.564} C_VEL
LIN {X 0,Y 531.044,Z 433.043,A -85,B 0,C 180,E1 -4191.536,E2 -4191.536} C_VEL
LIN {X 0,Y 531.262,Z 438.383,A -85,B 0,C 180,E1 -4193.465,E2 -4193.465} C_VEL
LIN {X 0,Y 531.17,Z 446.507,A -85,B 0,C 180,E1 -4196.467,E2 -4196.467} C_VEL
LIN {X 0,Y 531.107,Z 454.126,A -85,B 0,C 180,E1 -4199.331,E2 -4199.331} C_VEL
LIN {X 0,Y 531.032,Z 462.54,A -85,B 0,C 180,E1 -4202.464,E2 -4202.464} C_VEL
LIN {X 0,Y 530.954,Z 470.409,A -85,B 0,C 180,E1 -4205.357,E2 -4205.357} C_VEL
LIN {X 0,Y 530.887,Z 479.437,A -85,B 0,C 180,E1 -4208.65,E2 -4208.65} C_VEL
LIN {X 0,Y 530.768,Z 487.083,A -85,B 0,C 180,E1 -4211.47,E2 -4211.47} C_VEL
LIN {X 0,Y 530.692,Z 493.173,A -85,B 0,C 180,E1 -4213.704,E2 -4213.704} C_VEL
LIN {X 0,Y 533.16,Z 505.833,A -85,B 0,C 180,E1 -4214.036,E2 -4214.036} C_VEL
LIN {X 0,Y 532.991,Z 518.257,A -85,B 0,C 180,E1 -4214.397,E2 -4214.397} C_VEL
LIN {X 0,Y 532.729,Z 528.768,A -85,B 0,C 180,E1 -4214.799,E2 -4214.799} C_VEL
LIN {X 0,Y 532.544,Z 538.896,A -85,B 0,C 180,E1 -4215.282,E2 -4215.282} C_VEL
LIN {X 0,Y 532.226,Z 548.928,A -85,B 0,C 180,E1 -4215.859,E2 -4215.859} C_VEL
LIN {X 0,Y 531.964,Z 558.732,A -85,B 0,C 180,E1 -4216.534,E2 -4216.534} C_VEL
LIN {X 0,Y 531.657,Z 568.22,A -85,B 0,C 180,E1 -4217.304,E2 -4217.304} C_VEL
LIN {X 0,Y 531.412,Z 577.422,A -85,B 0,C 180,E1 -4218.183,E2 -4218.183} C_VEL
LIN {X 0,Y 531.221,Z 585.877,A -85,B 0,C 180,E1 -4219.132,E2 -4219.132} C_VEL
LIN {X 0,Y 530.929,Z 594.585,A -85,B 0,C 180,E1 -4220.283,E2 -4220.283} C_VEL
LIN {X 0,Y 530.744,Z 602.821,A -85,B 0,C 180,E1 -4221.624,E2 -4221.624} C_VEL
LIN {X 0,Y 530.589,Z 608.609,A -85,B 0,C 180,E1 -4222.77,E2 -4222.77} C_VEL
LIN {X 0,Y 530.54,Z 613.368,A -85,B 0,C 180,E1 -4223.916,E2 -4223.916} C_VEL
LIN {X 0,Y 530.452,Z 617.199,A -85,B 0,C 180,E1 -4225.059,E2 -4225.059} C_VEL
LIN {X 0,Y 530.498,Z 620.183,A -85,B 0,C 180,E1 -4226.201,E2 -4226.201} C_VEL
LIN {X 0,Y 530.453,Z 621.76,A -85,B 0,C 180,E1 -4226.961,E2 -4226.961} C_VEL
LIN {X 0,Y 530.359,Z 623.765,A -85,B 0,C 180,E1 -4228.48,E2 -4228.48} C_VEL
LIN {X 0,Y 530.342,Z 624.43,A -85,B 0,C 180,E1 -4229.999,E2 -4229.999} C_VEL
LIN {X 0,Y 530.341,Z 624.344,A -85,B 0,C 180,E1 -4230.758,E2 -4230.758} C_VEL
LIN {X 0,Y 530.409,Z 623.011,A -85,B 0,C 180,E1 -4232.277,E2 -4232.277} C_VEL
LIN {X 0,Y 530.451,Z 621.931,A -85,B 0,C 180,E1 -4233.037,E2 -4233.037} C_VEL
LIN {X 0,Y 530.449,Z 618.54,A -85,B 0,C 180,E1 -4234.559,E2 -4234.559} C_VEL
LIN {X 0,Y 530.559,Z 615.073,A -85,B 0,C 180,E1 -4235.701,E2 -4235.701} C_VEL
LIN {X 0,Y 530.573,Z 610.7,A -85,B 0,C 180,E1 -4236.846,E2 -4236.846} C_VEL
LIN {X 0,Y 530.683,Z 605.326,A -85,B 0,C 180,E1 -4237.992,E2 -4237.992} C_VEL
LIN {X 0,Y 530.827,Z 598.846,A -85,B 0,C 180,E1 -4239.141,E2 -4239.141} C_VEL
LIN {X 0,Y 530.983,Z 592.469,A -85,B 0,C 180,E1 -4240.099,E2 -4240.099} C_VEL
LIN {X 0,Y 531.219,Z 585.028,A -85,B 0,C 180,E1 -4241.059,E2 -4241.059} C_VEL
LIN {X 0,Y 531.415,Z 577.183,A -85,B 0,C 180,E1 -4241.931,E2 -4241.931} C_VEL
LIN {X 0,Y 531.679,Z 569.258,A -85,B 0,C 180,E1 -4242.694,E2 -4242.694} C_VEL
LIN {X 0,Y 531.932,Z 559.941,A -85,B 0,C 180,E1 -4243.465,E2 -4243.465} C_VEL
LIN {X 0,Y 532.173,Z 550.351,A -85,B 0,C 180,E1 -4244.14,E2 -4244.14} C_VEL
LIN {X 0,Y 532.516,Z 540.597,A -85,B 0,C 180,E1 -4244.717,E2 -4244.717} C_VEL
LIN {X 0,Y 532.684,Z 530.846,A -85,B 0,C 180,E1 -4245.201,E2 -4245.201} C_VEL
LIN {X 0,Y 532.915,Z 519.639,A -85,B 0,C 180,E1 -4245.647,E2 -4245.647} C_VEL
LIN {X 0,Y 533.128,Z 508.649,A -85,B 0,C 180,E1 -4245.981,E2 -4245.981} C_VEL
LIN {X 0,Y 533.042,Z 504.513,A -85,B 0,C 180,E1 -4246.092,E2 -4246.092} C_VEL
LIN {X 0,Y 530.681,Z 493.157,A -85,B 0,C 180,E1 -4246.393,E2 -4246.393} C_VEL
LIN {X 0,Y 530.805,Z 485.174,A -85,B 0,C 180,E1 -4249.329,E2 -4249.329} C_VEL
LIN {X 0,Y 530.921,Z 477.667,A -85,B 0,C 180,E1 -4252.086,E2 -4252.086} C_VEL
LIN {X 0,Y 530.955,Z 469.538,A -85,B 0,C 180,E1 -4255.059,E2 -4255.059} C_VEL
LIN {X 0,Y 531.029,Z 462.643,A -85,B 0,C 180,E1 -4257.593,E2 -4257.593} C_VEL
LIN {X 0,Y 531.083,Z 455.662,A -85,B 0,C 180,E1 -4260.188,E2 -4260.188} C_VEL
LIN {X 0,Y 531.11,Z 448.581,A -85,B 0,C 180,E1 -4262.855,E2 -4262.855} C_VEL
LIN {X 0,Y 531.209,Z 441.197,A -85,B 0,C 180,E1 -4265.599,E2 -4265.599} C_VEL
LIN {X 0,Y 531.213,Z 434.69,A -85,B 0,C 180,E1 -4267.965,E2 -4267.965} C_VEL
LIN {X 0,Y 531.083,Z 432.96,A -85,B 0,C 180,E1 -4268.669,E2 -4268.669} C_VEL
LIN {X 0,Y 531.002,Z 432.967,A -85,B 0,C 180,E1 -4271.433,E2 -4271.433} C_VEL
LIN {X 0,Y 530.982,Z 432.972,A -85,B 0,C 180,E1 -4274.546,E2 -4274.546} C_VEL
LIN {X 0,Y 530.983,Z 432.972,A -85,B 0,C 180,E1 -4277.832,E2 -4277.832} C_VEL
LIN {X 0,Y 530.998,Z 432.964,A -85,B 0,C 180,E1 -4280.557,E2 -4280.557} C_VEL
LIN {X 0,Y 530.966,Z 432.968,A -85,B 0,C 180,E1 -4283.841,E2 -4283.841} C_VEL
LIN {X 0,Y 530.992,Z 432.97,A -85,B 0,C 180,E1 -4286.493,E2 -4286.493} C_VEL
LIN {X 0,Y 530.974,Z 432.965,A -85,B 0,C 180,E1 -4289.352,E2 -4289.352} C_VEL
LIN {X 0,Y 531.009,Z 432.962,A -85,B 0,C 180,E1 -4292.404,E2 -4292.404} C_VEL
LIN {X 0,Y 531.001,Z 432.966,A -85,B 0,C 180,E1 -4294.942,E2 -4294.942} C_VEL
LIN {X 0,Y 530.982,Z 432.962,A -85,B 0,C 180,E1 -4297.893,E2 -4297.893} C_VEL
LIN {X 0,Y 530.988,Z 432.968,A -85,B 0,C 180,E1 -4300.677,E2 -4300.677} C_VEL
LIN {X 0,Y 530.984,Z 432.965,A -85,B 0,C 180,E1 -4303.071,E2 -4303.071} C_VEL
LIN {X 0,Y 531.009,Z 432.967,A -85,B 0,C 180,E1 -4305.435,E2 -4305.435} C_VEL
LIN {X 0,Y 531.042,Z 432.958,A -85,B 0,C 180,E1 -4308.55,E2 -4308.55} C_VEL
LIN {X 0,Y 531.052,Z 432.956,A -85,B 0,C 180,E1 -4311.629,E2 -4311.629} C_VEL
LIN {X 0,Y 531.135,Z 432.947,A -85,B 0,C 180,E1 -4314.685,E2 -4314.685} C_VEL
LIN {X 0,Y 531.13,Z 432.953,A -85,B 0,C 180,E1 -4317.725,E2 -4317.725} C_VEL
LIN {X 0,Y 531.146,Z 432.947,A -85,B 0,C 180,E1 -4320.758,E2 -4320.758} C_VEL
LIN {X 0,Y 531.102,Z 432.949,A -85,B 0,C 180,E1 -4323.034,E2 -4323.034} C_VEL
LIN {X 0,Y 531.076,Z 432.956,A -85,B 0,C 180,E1 -4326.077,E2 -4326.077} C_VEL
LIN {X 0,Y 531.028,Z 432.959,A -85,B 0,C 180,E1 -4329.138,E2 -4329.138} C_VEL
LIN {X 0,Y 531.031,Z 432.958,A -85,B 0,C 180,E1 -4332.225,E2 -4332.225} C_VEL
LIN {X 0,Y 530.986,Z 432.966,A -85,B 0,C 180,E1 -4335.35,E2 -4335.35} C_VEL
LIN {X 0,Y 531.006,Z 432.957,A -85,B 0,C 180,E1 -4337.723,E2 -4337.723} C_VEL
LIN {X 0,Y 530.994,Z 432.965,A -85,B 0,C 180,E1 -4340.938,E2 -4340.938} C_VEL
LIN {X 0,Y 530.97,Z 432.968,A -85,B 0,C 180,E1 -4344.225,E2 -4344.225} C_VEL
LIN {X 0,Y 531.003,Z 432.965,A -85,B 0,C 180,E1 -4346.744,E2 -4346.744} C_VEL
LIN {X 0,Y 530.991,Z 432.967,A -85,B 0,C 180,E1 -4349.322,E2 -4349.322} C_VEL
LIN {X 0,Y 530.972,Z 432.971,A -85,B 0,C 180,E1 -4352.104,E2 -4352.104} C_VEL
LIN {X 0,Y 530.983,Z 432.966,A -85,B 0,C 180,E1 -4354.855,E2 -4354.855} C_VEL
LIN {X 0,Y 530.958,Z 432.975,A -85,B 0,C 180,E1 -4357.508,E2 -4357.508} C_VEL
LIN {X 0,Y 531.002,Z 432.964,A -85,B 0,C 180,E1 -4360.431,E2 -4360.431} C_VEL
LIN {X 0,Y 530.961,Z 432.969,A -85,B 0,C 180,E1 -4363.495,E2 -4363.495} C_VEL
LIN {X 0,Y 530.952,Z 432.974,A -85,B 0,C 180,E1 -4366.506,E2 -4366.506} C_VEL
LIN {X 0,Y 531.021,Z 432.967,A -85,B 0,C 180,E1 -4369.572,E2 -4369.572} C_VEL
LIN {X 0,Y 530.964,Z 432.97,A -85,B 0,C 180,E1 -4372.578,E2 -4372.578} C_VEL
LIN {X 0,Y 531.025,Z 433.162,A -85,B 0,C 180,E1 -4375.141,E2 -4375.141} C_VEL
LIN {X 0,Y 532.25,Z 439.75,A -85,B 0,C 180,E1 -4377.224,E2 -4377.224} C_VEL
LIN {X 0,Y 532.336,Z 444.306,A -85,B 0,C 180,E1 -4378.569,E2 -4378.569} C_VEL
LIN {X 0,Y 531.964,Z 455.025,A -85,B 0,C 180,E1 -4381.602,E2 -4381.602} C_VEL
LIN {X 0,Y 531.639,Z 465.842,A -85,B 0,C 180,E1 -4384.557,E2 -4384.557} C_VEL
LIN {X 0,Y 531.354,Z 476.677,A -85,B 0,C 180,E1 -4387.446,E2 -4387.446} C_VEL
LIN {X 0,Y 531.153,Z 487.884,A -85,B 0,C 180,E1 -4390.314,E2 -4390.314} C_VEL
LIN {X 0,Y 531.001,Z 498.823,A -85,B 0,C 180,E1 -4393.073,E2 -4393.073} C_VEL
LIN {X 0,Y 530.957,Z 501.089,A -85,B 0,C 180,E1 -4393.64,E2 -4393.64} C_VEL
LIN {X 0,Y 533.227,Z 513.358,A -85,B 0,C 180,E1 -4393.933,E2 -4393.933} C_VEL
LIN {X 0,Y 532.973,Z 527.711,A -85,B 0,C 180,E1 -4394.326,E2 -4394.326} C_VEL
LIN {X 0,Y 532.675,Z 542.187,A -85,B 0,C 180,E1 -4394.897,E2 -4394.897} C_VEL
LIN {X 0,Y 532.37,Z 555.072,A -85,B 0,C 180,E1 -4395.572,E2 -4395.572} C_VEL
LIN {X 0,Y 531.993,Z 566.859,A -85,B 0,C 180,E1 -4396.342,E2 -4396.342} C_VEL
